C01819=1016.090,-13.127,392.870,165.816,56.691,160.189
C01820=1016.085,-13.376,392.883,165.813,56.699,160.190
C01821=1016.079,-13.625,392.895,165.811,56.706,160.191
C01822=1016.074,-13.876,392.908,165.808,56.714,160.192
C01823=1016.069,-14.125,392.920,165.806,56.722,160.192
C01824=1016.064,-14.374,392.933,165.803,56.729,160.193
C01825=1016.059,-14.625,392.945,165.801,56.737,160.194
C01826=1016.053,-14.874,392.957,165.797,56.744,160.195
C01827=1016.049,-15.123,392.970,165.795,56.752,160.195
C01828=1016.043,-15.373,392.982,165.792,56.760,160.196
C01829=1016.038,-15.623,392.994,165.790,56.767,160.197
C01830=1016.033,-15.873,393.007,165.787,56.775,160.198
C01831=1016.027,-16.122,393.019,165.784,56.782,160.198
C01832=1016.022,-16.372,393.031,165.782,56.790,160.199
C01833=1016.017,-16.621,393.043,165.779,56.797,160.200
C01834=1016.011,-16.871,393.055,165.776,56.805,160.201
C01835=1016.006,-17.121,393.067,165.773,56.813,160.202
C01836=1016.002,-17.371,393.080,165.771,56.821,160.202
C01837=1015.996,-17.621,393.091,165.769,56.828,160.203
C01838=1015.991,-17.870,393.104,165.766,56.836,160.204
C01839=1015.985,-18.120,393.116,165.764,56.844,160.205
C01840=1015.980,-18.369,393.127,165.760,56.852,160.206
C01841=1015.975,-18.619,393.140,165.758,56.859,160.207
C01842=1015.970,-18.869,393.151,165.755,56.867,160.207
C01843=1015.964,-19.118,393.163,165.753,56.875,160.208
C01844=1015.959,-19.368,393.175,165.751,56.882,160.209
C01845=1015.953,-19.618,393.188,165.747,56.890,160.210
C01846=1015.948,-19.868,393.199,165.744,56.897,160.210
C01847=1015.943,-20.117,393.211,165.742,56.905,160.211
C01848=1015.939,-20.367,393.223,165.739,56.913,160.212
C01849=1015.933,-20.616,393.235,165.737,56.920,160.213
C01850=1015.928,-20.867,393.247,165.734,56.928,160.214
C01851=1015.923,-21.116,393.259,165.732,56.936,160.215
C01852=1015.917,-21.392,393.273,165.729,56.944,160.215
C01853=1015.911,-21.670,393.286,165.726,56.952,160.216
C01854=1015.905,-21.946,393.299,165.722,56.961,160.217
C01855=1015.900,-22.223,393.312,165.719,56.969,160.218
C01856=1015.894,-22.472,393.324,165.717,56.977,160.219
C01857=1015.889,-22.722,393.336,165.714,56.984,160.219
C01858=1015.884,-22.972,393.348,165.712,56.992,160.220
C01859=1015.879,-23.222,393.360,165.709,56.999,160.221
C01860=1015.874,-23.471,393.371,165.707,57.007,160.222
C01861=1015.868,-23.721,393.383,165.704,57.014,160.222
C01862=1015.863,-23.970,393.395,165.701,57.022,160.223
C01863=1015.858,-24.220,393.407,165.699,57.029,160.224
C01864=1015.852,-24.470,393.419,165.696,57.037,160.225
C01865=1015.847,-24.719,393.431,165.693,57.044,160.225
C01866=1015.842,-24.969,393.443,165.690,57.052,160.226
C01867=1015.838,-25.219,393.455,165.688,57.060,160.227
C01868=1015.832,-25.468,393.467,165.685,57.067,160.227
C01869=1015.827,-25.718,393.478,165.682,57.074,160.228
C01870=1015.822,-25.968,393.490,165.680,57.082,160.229
C01871=1015.817,-26.217,393.502,165.677,57.089,160.230
C01872=1015.811,-26.468,393.514,165.675,57.097,160.230
C01873=1015.806,-26.717,393.526,165.672,57.104,160.231
C01874=1015.801,-26.967,393.537,165.669,57.111,160.232
C01875=1015.796,-27.216,393.549,165.667,57.119,160.233
C01876=1015.791,-27.466,393.561,165.664,57.126,160.233
C01877=1015.786,-27.715,393.573,165.662,57.134,160.234
C01878=1015.781,-27.965,393.584,165.659,57.141,160.235
C01879=1015.776,-28.215,393.596,165.655,57.149,160.235
C01880=1015.771,-28.465,393.607,165.653,57.156,160.236
C01881=1015.765,-28.714,393.618,165.651,57.164,160.237
C01882=1015.760,-28.963,393.630,165.648,57.172,160.238
C01883=1015.755,-29.213,393.642,165.645,57.179,160.238
C01884=1015.749,-29.464,393.653,165.643,57.187,160.239
C01885=1015.744,-29.714,393.665,165.639,57.195,160.240
C01886=1015.738,-29.963,393.676,165.637,57.202,160.241
C01887=1015.733,-30.213,393.687,165.634,57.209,160.241
C01888=1015.728,-30.463,393.699,165.632,57.217,160.242
C01889=1015.723,-30.712,393.711,165.629,57.225,160.243
C01890=1015.717,-30.961,393.722,165.627,57.232,160.244
C01891=1015.712,-31.211,393.733,165.624,57.239,160.245
C01892=1015.707,-31.461,393.745,165.621,57.248,160.245
C01893=1015.702,-31.711,393.756,165.618,57.255,160.246
C01894=1015.697,-31.961,393.768,165.615,57.262,160.247
C01895=1015.692,-32.210,393.779,165.613,57.270,160.247
C01896=1015.687,-32.460,393.790,165.611,57.278,160.248
C01897=1015.682,-32.710,393.801,165.608,57.285,160.249
C01898=1015.677,-32.959,393.813,165.605,57.292,160.250
C01899=1015.671,-33.209,393.824,165.602,57.299,160.250
C01900=1015.666,-33.459,393.835,165.600,57.307,160.251
C01901=1015.661,-33.709,393.847,165.597,57.315,160.252
C01902=1015.656,-33.958,393.858,165.594,57.322,160.252
C01903=1015.650,-34.208,393.869,165.591,57.330,160.253
C01904=1015.645,-34.458,393.881,165.589,57.337,160.254
C01905=1015.641,-34.707,393.892,165.586,57.345,160.255
C01906=1015.636,-34.957,393.903,165.583,57.352,160.255
C01907=1015.631,-35.206,393.915,165.581,57.359,160.256
C01908=1015.625,-35.456,393.926,165.578,57.366,160.257
C01909=1015.620,-35.706,393.937,165.576,57.374,160.257
C01910=1015.615,-35.955,393.948,165.573,57.381,160.258
C01911=1015.610,-36.205,393.960,165.570,57.389,160.259
C01912=1015.604,-36.455,393.971,165.567,57.396,160.259
C01913=1015.599,-36.705,393.982,165.565,57.403,160.260
C01914=1015.594,-36.954,393.994,165.562,57.410,160.261
C01915=1015.589,-37.204,394.005,165.560,57.418,160.262
C01916=1015.584,-37.445,394.015,165.557,57.425,160.262
C01917=1015.579,-37.685,394.027,165.554,57.432,160.263
C01918=1015.575,-37.925,394.037,165.551,57.439,160.263
C01919=1015.570,-38.166,394.048,165.549,57.447,160.264
C01920=1015.564,-38.406,394.059,165.547,57.453,160.265
C01921=1015.560,-38.647,394.070,165.544,57.460,160.266
C01922=1015.555,-38.887,394.080,165.541,57.467,160.266
C01923=1015.550,-39.128,394.092,165.538,57.474,160.267
C01924=1015.545,-39.378,394.102,165.536,57.482,160.267
C01925=1015.540,-39.627,394.113,165.533,57.489,160.268
C01926=1015.534,-39.877,394.124,165.531,57.497,160.269
C01927=1015.529,-40.127,394.136,165.528,57.504,160.269
C01928=1015.524,-40.376,394.146,165.526,57.512,160.270
C01929=1015.519,-40.626,394.157,165.523,57.519,160.271
C01930=1015.514,-40.875,394.168,165.520,57.526,160.272
C01931=1015.509,-41.126,394.179,165.517,57.535,160.272
C01932=1015.503,-41.375,394.190,165.514,57.542,160.273
C01933=1015.499,-41.624,394.201,165.512,57.549,160.274
C01934=1015.493,-41.874,394.212,165.509,57.556,160.274
C01935=1015.488,-42.124,394.222,165.507,57.564,160.275
C01936=1015.483,-42.374,394.233,165.504,57.571,160.276
C01937=1015.478,-42.624,394.244,165.501,57.579,160.277
C01938=1015.473,-42.873,394.254,165.498,57.586,160.277
C01939=1015.468,-43.123,394.266,165.496,57.593,160.278
C01940=1015.462,-43.373,394.276,165.493,57.601,160.279
C01941=1015.457,-43.623,394.288,165.490,57.608,160.279
C01942=1015.452,-43.872,394.298,165.488,57.615,160.280
C01943=1015.448,-44.122,394.309,165.484,57.623,160.280
C01944=1015.441,-44.416,394.322,165.481,57.632,160.281
C01945=1015.435,-44.711,394.335,165.478,57.640,160.282
C01946=1015.430,-45.005,394.347,165.475,57.649,160.283
C01947=1015.423,-45.299,394.360,165.472,57.657,160.284
C01948=1015.418,-45.549,394.370,165.470,57.665,160.284
C01949=1015.413,-45.798,394.381,165.467,57.672,160.285
C01950=1015.408,-46.048,394.392,165.464,57.679,160.286
C01951=1015.403,-46.298,394.403,165.462,57.687,160.286
C01952=1015.397,-46.548,394.413,165.459,57.694,160.287
C01953=1015.392,-46.797,394.424,165.456,57.701,160.288
C01954=1015.388,-47.047,394.435,165.454,57.708,160.288
C01955=1015.382,-47.297,394.445,165.451,57.715,160.289
C01956=1015.377,-47.546,394.457,165.448,57.722,160.290
C01957=1015.372,-47.796,394.467,165.445,57.729,160.290
C01958=1015.367,-48.046,394.478,165.443,57.737,160.291
C01959=1015.362,-48.295,394.488,165.440,57.744,160.292
C01960=1015.357,-48.545,394.499,165.437,57.751,160.292
C01961=1015.352,-48.795,394.510,165.434,57.758,160.293
C01962=1015.348,-49.045,394.520,165.432,57.766,160.294
C01963=1015.342,-49.294,394.531,165.429,57.773,160.294
C01964=1015.337,-49.544,394.542,165.426,57.780,160.295
C01965=1015.332,-49.793,394.552,165.423,57.787,160.295
C01966=1015.327,-50.044,394.563,165.420,57.794,160.296
C01967=1015.322,-50.293,394.574,165.418,57.802,160.297
C01968=1015.318,-50.543,394.584,165.415,57.809,160.297
C01969=1015.312,-50.792,394.595,165.412,57.816,160.298
C01970=1015.307,-51.043,394.606,165.409,57.823,160.298
C01971=1015.302,-51.292,394.616,165.407,57.830,160.299
C01972=1015.297,-51.542,394.626,165.404,57.838,160.300
C01973=1015.291,-51.792,394.637,165.402,57.845,160.300
C01974=1015.286,-52.041,394.646,165.399,57.853,160.301
C01975=1015.281,-52.291,394.657,165.396,57.860,160.302
C01976=1015.275,-52.541,394.667,165.394,57.868,160.303
C01977=1015.271,-52.791,394.677,165.391,57.875,160.303
C01978=1015.265,-53.041,394.687,165.388,57.882,160.304
C01979=1015.260,-53.290,394.697,165.386,57.889,160.305
C01980=1015.255,-53.566,394.708,165.383,57.898,160.305
C01981=1015.249,-53.842,394.720,165.380,57.906,160.306
C01982=1015.243,-54.118,394.730,165.376,57.914,160.306
C01983=1015.238,-54.394,394.742,165.374,57.922,160.307
C01984=1015.232,-54.644,394.752,165.371,57.929,160.308
C01985=1015.227,-54.894,394.762,165.367,57.936,160.308
C01986=1015.222,-55.144,394.772,165.365,57.944,160.309
C01987=1015.217,-55.394,394.782,165.362,57.951,160.310
C01988=1015.212,-55.643,394.792,165.359,57.958,160.310
C01989=1015.206,-55.894,394.802,165.357,57.966,160.311
C01990=1015.201,-56.143,394.812,165.354,57.973,160.312
C01991=1015.196,-56.393,394.822,165.351,57.980,160.312
C01992=1015.191,-56.642,394.833,165.349,57.987,160.313
C01993=1015.185,-56.892,394.843,165.346,57.995,160.314
C01994=1015.181,-57.141,394.853,165.343,58.002,160.314
C01995=1015.175,-57.391,394.863,165.341,58.009,160.315
C01996=1015.170,-57.641,394.873,165.338,58.016,160.315
C01997=1015.165,-57.891,394.883,165.335,58.023,160.316
C01998=1015.160,-58.140,394.893,165.333,58.031,160.317
C01999=1015.155,-58.391,394.904,165.330,58.038,160.317
C02000=1015.151,-58.640,394.913,165.327,58.045,160.318
C02001=1015.146,-58.890,394.923,165.324,58.052,160.318
C02002=1015.140,-59.140,394.933,165.321,58.059,160.319
C02003=1015.135,-59.389,394.943,165.319,58.067,160.320
C02004=1015.130,-59.639,394.953,165.316,58.074,160.320
C02005=1015.125,-59.889,394.963,165.314,58.081,160.321
C02006=1015.120,-60.139,394.973,165.311,58.088,160.322
C02007=1015.115,-60.388,394.983,165.308,58.096,160.322
C02008=1015.109,-60.638,394.993,165.305,58.103,160.323
C02009=1015.105,-60.888,395.003,165.302,58.110,160.323
C02010=1015.100,-61.137,395.013,165.299,58.117,160.324
C02011=1015.095,-61.388,395.022,165.298,58.123,160.325
C02012=1015.090,-61.637,395.032,165.295,58.130,160.325
C02013=1015.084,-61.887,395.042,165.292,58.138,160.326
C02014=1015.080,-62.137,395.052,165.289,58.145,160.326
C02015=1015.075,-62.386,395.062,165.286,58.152,160.327
C02016=1015.069,-62.636,395.072,165.284,58.159,160.327
C02017=1015.064,-62.886,395.082,165.281,58.166,160.328
C02018=1015.059,-63.136,395.092,165.278,58.173,160.328
C02019=1015.054,-63.385,395.102,165.275,58.180,160.329
C02020=1015.049,-63.635,395.111,165.272,58.187,160.330
C02021=1015.044,-63.885,395.121,165.270,58.194,160.330
C02022=1015.039,-64.135,395.131,165.268,58.201,160.331
C02023=1015.035,-64.384,395.140,165.265,58.208,160.331
C02024=1015.029,-64.634,395.151,165.262,58.215,160.332
C02025=1015.024,-64.884,395.160,165.259,58.222,160.333
C02026=1015.019,-65.133,395.170,165.257,58.229,160.333
C02027=1015.015,-65.384,395.180,165.254,58.236,160.334
C02028=1015.010,-65.633,395.190,165.251,58.243,160.334
C02029=1015.005,-65.883,395.200,165.249,58.249,160.335
C02030=1015.000,-66.133,395.210,165.246,58.256,160.335
C02031=1014.995,-66.382,395.220,165.243,58.263,160.336
C02032=1014.991,-66.632,395.229,165.240,58.270,160.336
C02033=1014.986,-66.882,395.239,165.238,58.278,160.337
C02034=1014.980,-67.132,395.249,165.235,58.285,160.338
C02035=1014.976,-67.381,395.259,165.232,58.291,160.338
C02036=1014.971,-67.631,395.268,165.230,58.298,160.339
C02037=1014.966,-67.882,395.278,165.227,58.305,160.339
C02038=1014.961,-68.131,395.288,165.224,58.312,160.340
C02039=1014.956,-68.380,395.297,165.221,58.319,160.340
C02040=1014.951,-68.630,395.307,165.219,58.325,160.341
C02041=1014.946,-68.880,395.317,165.216,58.332,160.341
C02042=1014.941,-69.130,395.327,165.213,58.339,160.342
C02043=1014.936,-69.379,395.336,165.210,58.345,160.342
C02044=1014.931,-69.656,395.347,165.208,58.353,160.343
C02045=1014.926,-69.934,395.358,165.205,58.360,160.343
C02046=1014.920,-70.210,395.368,165.201,58.368,160.344
C02047=1014.914,-70.488,395.379,165.199,58.376,160.345
C02048=1014.909,-70.738,395.388,165.196,58.382,160.345
C02049=1014.905,-70.987,395.398,165.193,58.389,160.346
C02050=1014.900,-71.237,395.408,165.191,58.396,160.346
C02051=1014.895,-71.487,395.417,165.188,58.402,160.347
C02052=1014.890,-71.737,395.427,165.185,58.409,160.347
C02053=1014.885,-71.987,395.436,165.183,58.416,160.348
C02054=1014.881,-72.236,395.446,165.180,58.422,160.348
C02055=1014.876,-72.486,395.456,165.177,58.430,160.349
C02056=1014.871,-72.736,395.465,165.175,58.435,160.349
C02057=1014.866,-72.986,395.475,165.172,58.443,160.350
C02058=1014.861,-73.235,395.485,165.169,58.450,160.350
C02059=1014.856,-73.485,395.494,165.166,58.456,160.350
C02060=1014.852,-73.735,395.504,165.164,58.463,160.351
C02061=1014.847,-73.985,395.513,165.161,58.469,160.352
C02062=1014.842,-74.234,395.523,165.159,58.476,160.352
C02063=1014.837,-74.483,395.532,165.156,58.482,160.353
C02064=1014.832,-74.734,395.542,165.153,58.489,160.353
C02065=1014.828,-74.984,395.551,165.149,58.496,160.353
C02066=1014.823,-75.234,395.561,165.148,58.502,160.354
C02067=1014.818,-75.484,395.570,165.145,58.509,160.355
C02068=1014.813,-75.733,395.579,165.142,58.517,160.355
C02069=1014.808,-75.983,395.588,165.139,58.523,160.355
C02070=1014.804,-76.233,395.597,165.137,58.530,160.356
C02071=1014.798,-76.482,395.606,165.134,58.537,160.357
C02072=1014.794,-76.732,395.615,165.131,58.543,160.357
///RCONF 1,0,0,0,1,0,0,0,0,0,0,0,0,0,0,0,0,0,0,0,0,0,0,0
C02073=1014.789,-76.982,395.624,165.128,58.550,160.358
C02074=1014.783,-77.232,395.634,165.126,58.557,160.358
C02075=1014.778,-77.482,395.643,165.123,58.563,160.359
C02076=1014.774,-77.732,395.652,165.120,58.570,160.359
C02077=1014.769,-77.981,395.662,165.117,58.577,160.359
C02078=1014.764,-78.231,395.670,165.115,58.583,160.360
C02079=1014.759,-78.481,395.680,165.113,58.591,160.361
C02080=1014.754,-78.730,395.689,165.109,58.597,160.361
C02081=1014.749,-78.980,395.698,165.107,58.604,160.362
C02082=1014.745,-79.230,395.707,165.104,58.610,160.362
C02083=1014.740,-79.480,395.716,165.101,58.617,160.363
C02084=1014.735,-79.729,395.725,165.098,58.624,160.363
C02085=1014.730,-79.979,395.734,165.096,58.630,160.364
C02086=1014.725,-80.229,395.743,165.093,58.637,160.364
C02087=1014.721,-80.479,395.752,165.090,58.644,160.364
C02088=1014.716,-80.729,395.761,165.089,58.650,160.365
C02089=1014.710,-80.979,395.769,165.085,58.657,160.365
C02090=1014.706,-81.229,395.778,165.082,58.664,160.366
C02091=1014.700,-81.478,395.788,165.080,58.671,160.367
C02092=1014.696,-81.728,395.797,165.076,58.677,160.367
C02093=1014.691,-81.977,395.805,165.075,58.684,160.368
C02094=1014.685,-82.227,395.814,165.072,58.691,160.368
C02095=1014.681,-82.477,395.823,165.068,58.698,160.368
C02096=1014.675,-82.727,395.831,165.066,58.705,160.369
C02097=1014.671,-82.977,395.840,165.063,58.711,160.369
C02098=1014.666,-83.227,395.849,165.061,58.718,160.370
C02099=1014.661,-83.477,395.858,165.058,58.725,160.371
C02100=1014.656,-83.726,395.866,165.056,58.731,160.371
C02101=1014.651,-83.976,395.875,165.053,58.738,160.372
C02102=1014.646,-84.226,395.884,165.050,58.745,160.372
C02103=1014.641,-84.476,395.892,165.047,58.752,160.372
C02104=1014.636,-84.726,395.902,165.045,58.758,160.373
C02105=1014.632,-84.975,395.910,165.042,58.765,160.373
C02106=1014.626,-85.225,395.918,165.038,58.771,160.374
C02107=1014.622,-85.475,395.927,165.037,58.778,160.374
C02108=1014.616,-85.754,395.937,165.033,58.786,160.375
C02109=1014.611,-86.033,395.947,165.030,58.793,160.375
C02110=1014.605,-86.312,395.956,165.028,58.800,160.376
C02111=1014.600,-86.591,395.966,165.024,58.807,160.376
C02112=1014.595,-86.841,395.975,165.022,58.814,160.377
C02113=1014.590,-87.091,395.983,165.019,58.821,160.377
C02114=1014.585,-87.341,395.991,165.015,58.827,160.377
C02115=1014.581,-87.590,396.000,165.014,58.834,160.378
C02116=1014.576,-87.840,396.008,165.010,58.840,160.378
C02117=1014.571,-88.090,396.017,165.009,58.847,160.379
C02118=1014.566,-88.340,396.026,165.005,58.853,160.379
C02119=1014.561,-88.590,396.034,165.002,58.860,160.380
C02120=1014.556,-88.840,396.044,165.000,58.866,160.380
C02121=1014.551,-89.089,396.052,164.997,58.873,160.381
C02122=1014.547,-89.339,396.061,164.995,58.879,160.381
C02123=1014.542,-89.589,396.068,164.992,58.886,160.382
C02124=1014.537,-89.839,396.077,164.990,58.892,160.382
C02125=1014.532,-90.089,396.086,164.986,58.898,160.382
C02126=1014.527,-90.338,396.094,164.983,58.905,160.383
C02127=1014.523,-90.588,396.103,164.981,58.911,160.383
C02128=1014.518,-90.837,396.112,164.978,58.918,160.384
C02129=1014.513,-91.088,396.119,164.976,58.924,160.384
C02130=1014.508,-91.338,396.129,164.973,58.930,160.384
C02131=1014.504,-91.587,396.137,164.971,58.937,160.385
C02132=1014.499,-91.837,396.146,164.968,58.943,160.385
C02133=1014.494,-92.087,396.154,164.965,58.949,160.386
C02134=1014.489,-92.337,396.162,164.962,58.956,160.386
C02135=1014.485,-92.586,396.171,164.960,58.962,160.387
C02136=1014.480,-92.836,396.179,164.957,58.969,160.387
C02137=1014.475,-93.086,396.188,164.955,58.975,160.388
C02138=1014.470,-93.336,396.196,164.951,58.981,160.388
C02139=1014.465,-93.585,396.204,164.949,58.987,160.388
C02140=1014.461,-93.835,396.213,164.947,58.993,160.389
C02141=1014.456,-94.086,396.221,164.944,59.000,160.389
C02142=1014.452,-94.335,396.230,164.941,59.006,160.389
C02143=1014.447,-94.585,396.238,164.938,59.012,160.390
C02144=1014.442,-94.834,396.247,164.936,59.018,160.390
C02145=1014.438,-95.084,396.255,164.933,59.025,160.391
C02146=1014.433,-95.334,396.263,164.931,59.031,160.391
C02147=1014.427,-95.584,396.272,164.928,59.037,160.392
C02148=1014.423,-95.834,396.280,164.925,59.044,160.392
C02149=1014.418,-96.083,396.288,164.923,59.050,160.392
C02150=1014.414,-96.334,396.297,164.920,59.056,160.393
C02151=1014.410,-96.583,396.305,164.917,59.062,160.393
C02152=1014.404,-96.833,396.313,164.915,59.068,160.393
C02153=1014.400,-97.083,396.322,164.912,59.074,160.394
C02154=1014.395,-97.333,396.330,164.909,59.080,160.394
C02155=1014.391,-97.583,396.339,164.907,59.086,160.395
C02156=1014.386,-97.833,396.346,164.903,59.092,160.394
C02157=1014.381,-98.082,396.355,164.901,59.098,160.395
C02158=1014.376,-98.332,396.362,164.898,59.105,160.396
C02159=1014.372,-98.582,396.371,164.896,59.111,160.396
C02160=1014.367,-98.832,396.379,164.893,59.118,160.396
C02161=1014.362,-99.082,396.387,164.890,59.124,160.397
C02162=1014.357,-99.332,396.395,164.888,59.130,160.397
C02163=1014.353,-99.581,396.403,164.885,59.136,160.397
C02164=1014.348,-99.831,396.411,164.883,59.142,160.398
C02165=1014.343,-100.081,396.418,164.879,59.149,160.398
C02166=1014.338,-100.331,396.427,164.877,59.155,160.399
C02167=1014.334,-100.580,396.434,164.874,59.161,160.399
C02168=1014.328,-100.830,396.443,164.872,59.167,160.399
C02169=1014.324,-101.081,396.451,164.869,59.173,160.400
C02170=1014.320,-101.330,396.459,164.866,59.179,160.400
C02171=1014.315,-101.580,396.467,164.864,59.185,160.400
C02172=1014.310,-101.861,396.475,164.861,59.193,160.401
C02173=1014.304,-102.142,396.484,164.858,59.199,160.401
C02174=1014.299,-102.423,396.493,164.855,59.206,160.402
C02175=1014.293,-102.704,396.502,164.852,59.213,160.402
C02176=1014.288,-102.953,396.510,164.850,59.219,160.402
C02177=1014.284,-103.204,396.518,164.846,59.225,160.403
C02178=1014.279,-103.453,396.525,164.844,59.231,160.403
C02179=1014.275,-103.703,396.534,164.842,59.237,160.404
C02180=1014.270,-103.953,396.542,164.838,59.244,160.404
C02181=1014.265,-104.203,396.550,164.836,59.250,160.404
C02182=1014.261,-104.453,396.557,164.834,59.256,160.405
C02183=1014.256,-104.703,396.565,164.831,59.262,160.405
C02184=1014.251,-104.952,396.573,164.828,59.267,160.405
C02185=1014.246,-105.203,396.581,164.826,59.273,160.405
C02186=1014.242,-105.452,396.588,164.822,59.280,160.406
C02187=1014.237,-105.702,396.596,164.820,59.286,160.406
C02188=1014.232,-105.952,396.604,164.818,59.292,160.407
C02189=1014.228,-106.201,396.611,164.816,59.298,160.407
C02190=1014.223,-106.452,396.619,164.812,59.304,160.407
C02191=1014.218,-106.701,396.627,164.809,59.310,160.407
C02192=1014.213,-106.951,396.635,164.807,59.316,160.408
C02193=1014.209,-107.201,396.642,164.805,59.322,160.408
C02194=1014.204,-107.451,396.650,164.801,59.327,160.408
C02195=1014.200,-107.701,396.657,164.799,59.333,160.409
C02196=1014.195,-107.950,396.665,164.797,59.339,160.409
C02197=1014.190,-108.201,396.673,164.794,59.345,160.410
C02198=1014.186,-108.450,396.681,164.792,59.351,160.410
C02199=1014.181,-108.700,396.689,164.788,59.357,160.410
C02200=1014.176,-108.950,396.696,164.786,59.363,160.410
C02201=1014.172,-109.199,396.703,164.784,59.369,160.411
C02202=1014.167,-109.450,396.711,164.781,59.375,160.411
C02203=1014.163,-109.699,396.719,164.778,59.381,160.411
C02204=1014.158,-109.950,396.726,164.775,59.387,160.412
C02205=1014.153,-110.199,396.733,164.773,59.393,160.412
C02206=1014.148,-110.448,396.741,164.771,59.399,160.413
C02207=1014.143,-110.699,396.748,164.767,59.405,160.413
C02208=1014.139,-110.948,396.756,164.765,59.411,160.413
C02209=1014.135,-111.198,396.763,164.763,59.417,160.413
C02210=1014.130,-111.448,396.771,164.760,59.422,160.414
C02211=1014.125,-111.698,396.778,164.757,59.428,160.414
C02212=1014.121,-111.948,396.786,164.755,59.434,160.415
C02213=1014.115,-112.198,396.793,164.751,59.440,160.414
C02214=1014.111,-112.447,396.800,164.749,59.446,160.415
C02215=1014.107,-112.697,396.808,164.747,59.452,160.415
C02216=1014.102,-112.947,396.815,164.744,59.457,160.415
C02217=1014.097,-113.197,396.823,164.742,59.463,160.416
C02218=1014.093,-113.447,396.830,164.739,59.468,160.416
C02219=1014.089,-113.697,396.837,164.737,59.474,160.416
C02220=1014.084,-113.947,396.845,164.734,59.480,160.417
C02221=1014.080,-114.197,396.852,164.732,59.486,160.417
C02222=1014.075,-114.446,396.859,164.728,59.492,160.417
C02223=1014.070,-114.696,396.867,164.726,59.497,160.417
C02224=1014.065,-114.946,396.874,164.723,59.503,160.418
C02225=1014.061,-115.196,396.881,164.720,59.509,160.418
C02226=1014.056,-115.445,396.889,164.718,59.515,160.418
C02227=1014.051,-115.696,396.895,164.715,59.520,160.419
C02228=1014.047,-115.946,396.903,164.713,59.526,160.419
C02229=1014.042,-116.195,396.910,164.710,59.531,160.419
C02230=1014.038,-116.445,396.918,164.708,59.537,160.420
C02231=1014.032,-116.695,396.925,164.705,59.543,160.420
C02232=1014.028,-116.945,396.931,164.703,59.549,160.420
C02233=1014.024,-117.195,396.939,164.700,59.554,160.420
C02234=1014.020,-117.444,396.946,164.698,59.560,160.421
C02235=1014.014,-117.694,396.953,164.695,59.565,160.421
C02236=1014.009,-117.976,396.961,164.692,59.572,160.421
C02237=1014.004,-118.257,396.969,164.689,59.578,160.421
C02238=1013.999,-118.538,396.977,164.686,59.584,160.422
C02239=1013.994,-118.819,396.985,164.683,59.591,160.422
C02240=1013.989,-119.069,396.992,164.681,59.597,160.422
C02241=1013.985,-119.320,396.999,164.678,59.602,160.423
C02242=1013.980,-119.569,397.006,164.676,59.608,160.423
C02243=1013.975,-119.819,397.014,164.673,59.613,160.423
C02244=1013.971,-120.069,397.020,164.670,59.619,160.423
C02245=1013.966,-120.318,397.027,164.668,59.625,160.424
C02246=1013.962,-120.568,397.034,164.665,59.630,160.424
C02247=1013.957,-120.819,397.041,164.663,59.636,160.424
C02248=1013.953,-121.068,397.049,164.660,59.641,160.424
C02249=1013.948,-121.318,397.055,164.657,59.647,160.425
C02250=1013.944,-121.568,397.062,164.655,59.653,160.425
C02251=1013.939,-121.818,397.070,164.652,59.658,160.425
C02252=1013.935,-122.068,397.076,164.649,59.663,160.425
C02253=1013.930,-122.317,397.083,164.648,59.669,160.426
C02254=1013.926,-122.567,397.090,164.645,59.674,160.426
C02255=1013.921,-122.817,397.097,164.643,59.679,160.426
C02256=1013.916,-123.067,397.105,164.640,59.685,160.426
C02257=1013.912,-123.317,397.111,164.638,59.691,160.427
C02258=1013.907,-123.567,397.118,164.635,59.696,160.427
C02259=1013.903,-123.817,397.125,164.632,59.701,160.427
C02260=1013.898,-124.066,397.132,164.629,59.707,160.427
C02261=1013.894,-124.317,397.138,164.627,59.711,160.428
C02262=1013.889,-124.566,397.146,164.625,59.717,160.428
C02263=1013.885,-124.816,397.152,164.622,59.723,160.428
C02264=1013.880,-125.066,397.159,164.619,59.728,160.428
C02265=1013.876,-125.316,397.166,164.617,59.733,160.428
C02266=1013.871,-125.565,397.173,164.614,59.739,160.429
C02267=1013.867,-125.816,397.179,164.612,59.745,160.429
C02268=1013.862,-126.066,397.185,164.609,59.750,160.429
C02269=1013.858,-126.315,397.193,164.607,59.755,160.429
C02270=1013.853,-126.565,397.199,164.604,59.760,160.430
C02271=1013.849,-126.815,397.206,164.602,59.766,160.430
C02272=1013.844,-127.065,397.212,164.599,59.771,160.430
C02273=1013.840,-127.315,397.219,164.596,59.777,160.430
C02274=1013.835,-127.564,397.226,164.595,59.782,160.431
C02275=1013.831,-127.814,397.233,164.592,59.787,160.431
C02276=1013.826,-128.064,397.239,164.589,59.792,160.431
C02277=1013.822,-128.314,397.246,164.586,59.797,160.431
C02278=1013.818,-128.563,397.253,164.584,59.802,160.431
C02279=1013.813,-128.813,397.261,164.582,59.806,160.431
C02280=1013.810,-129.062,397.270,164.580,59.810,160.431
C02281=1013.807,-129.312,397.279,164.578,59.813,160.431
C02282=1013.804,-129.562,397.288,164.575,59.817,160.431
C02283=1013.802,-129.812,397.299,164.572,59.819,160.431
C02284=1013.799,-130.061,397.310,164.570,59.821,160.430
C02285=1013.798,-130.311,397.321,164.568,59.821,160.430
C02286=1013.797,-130.560,397.334,164.566,59.822,160.429
C02287=1013.796,-130.810,397.347,164.563,59.822,160.429
C02288=1013.795,-131.060,397.360,164.561,59.822,160.428
C02289=1013.795,-131.310,397.374,164.560,59.822,160.427
C02290=1013.794,-131.559,397.388,164.557,59.821,160.426
C02291=1013.795,-131.809,397.403,164.555,59.819,160.425
C02292=1013.796,-132.059,397.419,164.552,59.817,160.424
C02293=1013.797,-132.308,397.435,164.551,59.814,160.423
C02294=1013.798,-132.558,397.452,164.549,59.811,160.422
C02295=1013.800,-132.807,397.470,164.547,59.808,160.421
C02296=1013.802,-133.057,397.488,164.545,59.803,160.419
C02297=1013.804,-133.307,397.507,164.543,59.799,160.418
C02298=1013.807,-133.556,397.527,164.541,59.794,160.416
C02299=1013.810,-133.806,397.547,164.539,59.788,160.415
C02300=1013.579,-133.832,397.130,164.519,60.110,160.468
C02301=1013.576,-133.583,397.110,164.521,60.115,160.470
C02302=1013.574,-133.333,397.091,164.523,60.119,160.471
C02303=1013.571,-133.083,397.072,164.526,60.124,160.473
C02304=1013.570,-132.833,397.053,164.527,60.128,160.474
C02305=1013.568,-132.584,397.035,164.530,60.131,160.475
C02306=1013.566,-132.334,397.018,164.530,60.134,160.476
C02307=1013.565,-132.084,397.003,164.533,60.137,160.478
C02308=1013.564,-131.835,396.986,164.535,60.139,160.478
C02309=1013.564,-131.585,396.971,164.538,60.140,160.480
C02310=1013.564,-131.336,396.957,164.539,60.142,160.480
C02311=1013.565,-131.086,396.943,164.541,60.142,160.481
C02312=1013.565,-130.836,396.929,164.544,60.142,160.482
C02313=1013.566,-130.587,396.917,164.545,60.142,160.482
C02314=1013.568,-130.338,396.904,164.548,60.141,160.483
C02315=1013.569,-130.088,396.893,164.550,60.140,160.483
C02316=1013.571,-129.838,396.881,164.552,60.138,160.484
C02317=1013.574,-129.588,396.871,164.554,60.137,160.484
C02318=1013.576,-129.338,396.862,164.558,60.134,160.485
C02319=1013.579,-129.088,396.852,164.560,60.131,160.485
C02320=1013.583,-128.839,396.844,164.562,60.127,160.485
C02321=1013.586,-128.590,396.836,164.563,60.123,160.484
C02322=1013.590,-128.340,396.829,164.567,60.119,160.485
C02323=1013.595,-128.090,396.822,164.568,60.114,160.484
C02324=1013.600,-127.841,396.815,164.571,60.109,160.484
C02325=1013.604,-127.591,396.809,164.574,60.104,160.484
C02326=1013.608,-127.342,396.802,164.576,60.099,160.484
C02327=1013.613,-127.092,396.796,164.579,60.094,160.484
C02328=1013.617,-126.842,396.789,164.581,60.089,160.484
C02329=1013.622,-126.592,396.782,164.584,60.084,160.483
C02330=1013.626,-126.342,396.776,164.587,60.078,160.483
C02331=1013.631,-126.092,396.770,164.588,60.073,160.483
C02332=1013.635,-125.842,396.762,164.591,60.068,160.483
C02333=1013.640,-125.593,396.756,164.594,60.063,160.483
C02334=1013.644,-125.342,396.749,164.597,60.058,160.483
C02335=1013.648,-125.093,396.742,164.598,60.053,160.482
C02336=1013.653,-124.843,396.736,164.601,60.047,160.482
C02337=1013.658,-124.593,396.728,164.604,60.042,160.482
C02338=1013.662,-124.343,396.722,164.606,60.037,160.482
C02339=1013.667,-124.093,396.715,164.608,60.032,160.481
C02340=1013.671,-123.843,396.708,164.611,60.027,160.481
C02341=1013.677,-123.593,396.701,164.613,60.022,160.481
C02342=1013.681,-123.343,396.694,164.616,60.016,160.481
C02343=1013.685,-123.093,396.687,164.619,60.011,160.481
C02344=1013.690,-122.843,396.681,164.621,60.006,160.481
C02345=1013.694,-122.594,396.673,164.623,60.001,160.480
C02346=1013.698,-122.343,396.667,164.626,59.996,160.480
C02347=1013.703,-122.094,396.660,164.629,59.990,160.480
C02348=1013.707,-121.844,396.653,164.632,59.985,160.480
C02349=1013.712,-121.594,396.646,164.633,59.980,160.479
C02350=1013.716,-121.344,396.640,164.636,59.975,160.479
C02351=1013.721,-121.095,396.632,164.638,59.969,160.479
C02352=1013.725,-120.845,396.625,164.641,59.963,160.479
C02353=1013.731,-120.594,396.619,164.644,59.958,160.479
C02354=1013.735,-120.345,396.611,164.646,59.953,160.478
C02355=1013.739,-120.095,396.604,164.648,59.948,160.478
C02356=1013.744,-119.845,396.598,164.651,59.943,160.478
C02357=1013.748,-119.596,396.590,164.654,59.937,160.478
C02358=1013.752,-119.345,396.584,164.656,59.931,160.477
C02359=1013.757,-119.096,396.576,164.659,59.926,160.477
C02360=1013.762,-118.846,396.569,164.662,59.921,160.477
C02361=1013.766,-118.565,396.562,164.664,59.915,160.477
C02362=1013.772,-118.283,396.553,164.667,59.908,160.476
C02363=1013.778,-118.002,396.546,164.670,59.903,160.476
C02364=1013.783,-117.721,396.537,164.673,59.896,160.476
C02365=1013.787,-117.471,396.530,164.675,59.891,160.476
C02366=1013.792,-117.222,396.523,164.677,59.885,160.475
C02367=1013.796,-116.972,396.517,164.680,59.880,160.475
C02368=1013.800,-116.722,396.509,164.683,59.875,160.475
C02369=1013.805,-116.472,396.501,164.685,59.869,160.475
C02370=1013.810,-116.222,396.494,164.688,59.863,160.474
C02371=1013.815,-115.972,396.488,164.690,59.858,160.474
C02372=1013.819,-115.723,396.481,164.693,59.853,160.474
C02373=1013.823,-115.473,396.473,164.695,59.847,160.474
C02374=1013.828,-115.223,396.465,164.698,59.841,160.473
C02375=1013.833,-114.973,396.459,164.700,59.835,160.473
C02376=1013.837,-114.723,396.452,164.703,59.830,160.473
C02377=1013.842,-114.474,396.444,164.706,59.825,160.473
C02378=1013.847,-114.223,396.437,164.708,59.819,160.472
C02379=1013.851,-113.974,396.429,164.711,59.813,160.472
C02380=1013.855,-113.724,396.422,164.714,59.808,160.472
C02381=1013.860,-113.475,396.415,164.716,59.802,160.471
C02382=1013.865,-113.224,396.408,164.719,59.797,160.471
C02383=1013.869,-112.974,396.401,164.722,59.791,160.471
C02384=1013.874,-112.724,396.393,164.724,59.785,160.471
C02385=1013.878,-112.475,396.386,164.727,59.780,160.471
C02386=1013.883,-112.224,396.378,164.729,59.774,160.470
C02387=1013.887,-111.975,396.371,164.732,59.769,160.470
C02388=1013.892,-111.725,396.363,164.734,59.763,160.469
C02389=1013.896,-111.475,396.356,164.737,59.757,160.469
C02390=1013.902,-111.225,396.349,164.739,59.751,160.469
C02391=1013.906,-110.976,396.341,164.742,59.746,160.469
C02392=1013.911,-110.726,396.334,164.744,59.740,160.468
C02393=1013.916,-110.476,396.326,164.747,59.735,160.468
C02394=1013.920,-110.226,396.319,164.749,59.729,160.468
C02395=1013.924,-109.977,396.311,164.751,59.723,160.468
C02396=1013.929,-109.726,396.304,164.754,59.717,160.467
C02397=1013.934,-109.477,396.296,164.756,59.712,160.467
C02398=1013.939,-109.227,396.289,164.760,59.705,160.467
C02399=1013.944,-108.977,396.282,164.763,59.700,160.467
C02400=1013.948,-108.727,396.274,164.765,59.694,160.466
C02401=1013.952,-108.478,396.267,164.767,59.688,160.466
C02402=1013.957,-108.227,396.259,164.770,59.683,160.465
C02403=1013.962,-107.978,396.252,164.772,59.677,160.465
C02404=1013.967,-107.727,396.244,164.775,59.671,160.465
C02405=1013.971,-107.478,396.236,164.777,59.665,160.464
C02406=1013.975,-107.228,396.229,164.780,59.659,160.464
C02407=1013.980,-106.978,396.221,164.783,59.654,160.464
C02408=1013.985,-106.728,396.214,164.785,59.648,160.464
C02409=1013.990,-106.478,396.205,164.788,59.642,160.463
C02410=1013.994,-106.229,396.198,164.790,59.636,160.463
C02411=1013.999,-105.979,396.191,164.792,59.630,160.462
C02412=1014.004,-105.729,396.183,164.795,59.625,160.462
C02413=1014.008,-105.479,396.175,164.798,59.619,160.462
C02414=1014.013,-105.229,396.168,164.801,59.612,160.462
C02415=1014.018,-104.980,396.159,164.803,59.607,160.461
C02416=1014.022,-104.729,396.151,164.806,59.601,160.461
C02417=1014.026,-104.480,396.144,164.808,59.595,160.461
C02418=1014.031,-104.230,396.136,164.812,59.589,160.461
C02419=1014.036,-103.980,396.128,164.814,59.583,160.460
C02420=1014.040,-103.731,396.120,164.816,59.577,160.460
C02421=1014.045,-103.480,396.113,164.818,59.571,160.459
C02422=1014.049,-103.231,396.105,164.821,59.566,160.459
C02423=1014.055,-102.981,396.097,164.824,59.560,160.459
C02424=1014.059,-102.731,396.089,164.827,59.554,160.458
C02425=1014.065,-102.450,396.080,164.830,59.547,160.458
C02426=1014.070,-102.169,396.072,164.832,59.540,160.458
C02427=1014.075,-101.889,396.063,164.836,59.533,160.457
C02428=1014.081,-101.607,396.054,164.839,59.527,160.457
C02429=1014.084,-101.357,396.046,164.841,59.521,160.457
C02430=1014.089,-101.107,396.038,164.843,59.515,160.456
C02431=1014.094,-100.858,396.030,164.846,59.509,160.456
C02432=1014.099,-100.608,396.022,164.849,59.502,160.455
C02433=1014.103,-100.358,396.015,164.851,59.496,160.455
C02434=1014.109,-100.108,396.006,164.854,59.491,160.455
C02435=1014.113,-99.859,395.999,164.857,59.485,160.455
C02436=1014.118,-99.609,395.990,164.859,59.478,160.454
C02437=1014.123,-99.359,395.983,164.861,59.472,160.454
C02438=1014.128,-99.109,395.975,164.865,59.466,160.453
C02439=1014.132,-98.859,395.966,164.867,59.460,160.453
C02440=1014.136,-98.609,395.959,164.869,59.454,160.452
C02441=1014.141,-98.359,395.951,164.872,59.447,160.452
C02442=1014.146,-98.110,395.943,164.875,59.441,160.452
C02443=1014.151,-97.860,395.935,164.878,59.435,160.451
C02444=1014.156,-97.610,395.926,164.880,59.429,160.451
C02445=1014.160,-97.360,395.918,164.883,59.424,160.451
C02446=1014.165,-97.110,395.910,164.885,59.418,160.450
C02447=1014.169,-96.861,395.901,164.888,59.411,160.450
C02448=1014.174,-96.611,395.893,164.891,59.405,160.450
C02449=1014.179,-96.361,395.884,164.893,59.399,160.449
C02450=1014.183,-96.111,395.877,164.896,59.393,160.449
C02451=1014.188,-95.861,395.868,164.898,59.387,160.448
C02452=1014.193,-95.611,395.859,164.901,59.381,160.448
C02453=1014.197,-95.362,395.852,164.903,59.375,160.448
C02454=1014.202,-95.112,395.844,164.907,59.369,160.448
C02455=1014.207,-94.862,395.834,164.909,59.363,160.447
C02456=1014.211,-94.612,395.827,164.911,59.357,160.447
C02457=1014.216,-94.362,395.818,164.914,59.350,160.446
C02458=1014.221,-94.113,395.809,164.917,59.344,160.446
C02459=1014.225,-93.863,395.802,164.920,59.338,160.446
C02460=1014.230,-93.613,395.793,164.922,59.332,160.445
C02461=1014.235,-93.363,395.785,164.924,59.326,160.445
C02462=1014.239,-93.113,395.777,164.928,59.320,160.445
C02463=1014.244,-92.864,395.768,164.930,59.314,160.444
C02464=1014.249,-92.614,395.760,164.933,59.307,160.444
C02465=1014.253,-92.365,395.751,164.935,59.301,160.443
C02466=1014.258,-92.114,395.743,164.937,59.295,160.443
C02467=1014.263,-91.864,395.734,164.941,59.289,160.443
C02468=1014.268,-91.614,395.725,164.943,59.283,160.442
C02469=1014.273,-91.365,395.717,164.946,59.276,160.442
C02470=1014.277,-91.115,395.709,164.948,59.269,160.441
C02471=1014.282,-90.865,395.701,164.951,59.263,160.441
C02472=1014.286,-90.616,395.692,164.953,59.257,160.440
C02473=1014.291,-90.366,395.683,164.957,59.251,160.440
C02474=1014.296,-90.116,395.676,164.959,59.245,160.440
C02475=1014.301,-89.866,395.666,164.962,59.238,160.439
C02476=1014.306,-89.617,395.658,164.964,59.232,160.439
C02477=1014.310,-89.367,395.649,164.967,59.225,160.438
C02478=1014.315,-89.117,395.641,164.969,59.219,160.438
C02479=1014.320,-88.867,395.633,164.973,59.212,160.438
C02480=1014.325,-88.617,395.624,164.975,59.206,160.437
C02481=1014.329,-88.368,395.616,164.977,59.199,160.437
C02482=1014.334,-88.118,395.607,164.980,59.193,160.436
C02483=1014.339,-87.868,395.598,164.983,59.187,160.436
C02484=1014.344,-87.618,395.590,164.985,59.181,160.435
C02485=1014.349,-87.367,395.581,164.988,59.174,160.435
C02486=1014.353,-87.118,395.573,164.990,59.168,160.434
C02487=1014.358,-86.868,395.564,164.993,59.161,160.434
C02488=1014.363,-86.619,395.556,164.996,59.154,160.434
C02489=1014.368,-86.340,395.546,164.999,59.148,160.433
C02490=1014.374,-86.060,395.536,165.002,59.140,160.433
C02491=1014.380,-85.782,395.527,165.005,59.133,160.432
C02492=1014.385,-85.503,395.517,165.008,59.126,160.432
C02493=1014.390,-85.253,395.509,165.010,59.119,160.431
C02494=1014.395,-85.003,395.500,165.013,59.112,160.431
C02495=1014.400,-84.754,395.491,165.016,59.105,160.430
C02496=1014.404,-84.504,395.482,165.018,59.099,160.430
C02497=1014.409,-84.255,395.474,165.022,59.093,160.429
C02498=1014.414,-84.005,395.465,165.023,59.086,160.429
C02499=1014.419,-83.755,395.457,165.026,59.080,160.428
C02500=1014.424,-83.505,395.448,165.029,59.072,160.428
C02501=1014.429,-83.255,395.439,165.031,59.066,160.427
C02502=1014.434,-83.005,395.431,165.034,59.059,160.427
C02503=1014.438,-82.755,395.422,165.037,59.053,160.427
C02504=1014.444,-82.506,395.413,165.040,59.046,160.426
C02505=1014.449,-82.256,395.405,165.042,59.040,160.425
C02506=1014.453,-82.006,395.395,165.045,59.033,160.425
C02507=1014.459,-81.756,395.387,165.048,59.026,160.425
C02508=1014.463,-81.507,395.378,165.050,59.019,160.424
C02509=1014.468,-81.257,395.370,165.053,59.012,160.423
C02510=1014.472,-81.007,395.361,165.056,59.006,160.423
C02511=1014.478,-80.757,395.352,165.059,58.999,160.422
C02512=1014.483,-80.508,395.344,165.061,58.993,160.422
C02513=1014.488,-80.258,395.335,165.063,58.985,160.421
C02514=1014.492,-80.008,395.326,165.067,58.979,160.421
C02515=1014.497,-79.758,395.317,165.068,58.972,160.420
C02516=1014.502,-79.508,395.308,165.072,58.966,160.420
C02517=1014.507,-79.259,395.298,165.074,58.959,160.420
C02518=1014.511,-79.008,395.289,165.077,58.953,160.419
C02519=1014.516,-78.759,395.281,165.080,58.946,160.419
C02520=1014.521,-78.509,395.272,165.083,58.939,160.418
C02521=1014.526,-78.259,395.262,165.085,58.933,160.418
C02522=1014.531,-78.010,395.253,165.088,58.926,160.417
C02523=1014.536,-77.760,395.244,165.091,58.920,160.417
C02524=1014.540,-77.510,395.235,165.093,58.913,160.416
C02525=1014.546,-77.260,395.226,165.095,58.906,160.416
C02526=1014.551,-77.010,395.217,165.099,58.899,160.415
C02527=1014.555,-76.760,395.207,165.100,58.893,160.415
C02528=1014.560,-76.510,395.198,165.104,58.886,160.414
C02529=1014.565,-76.261,395.189,165.106,58.879,160.414
C02530=1014.570,-76.011,395.180,165.110,58.873,160.413
C02531=1014.575,-75.761,395.170,165.111,58.866,160.413
C02532=1014.580,-75.511,395.162,165.114,58.859,160.412
///RCONF 1,0,0,0,0,0,0,0,0,0,0,0,0,0,0,0,0,0,0,0,0,0,0,0
C02533=1014.585,-75.261,395.153,165.117,58.852,160.412
C02534=1014.589,-75.012,395.143,165.120,58.845,160.411
C02535=1014.595,-74.762,395.134,165.122,58.838,160.410
C02536=1014.599,-74.512,395.125,165.125,58.832,160.410
C02537=1014.604,-74.263,395.116,165.128,58.825,160.410
C02538=1014.609,-74.013,395.106,165.130,58.819,160.409
C02539=1014.614,-73.763,395.096,165.133,58.812,160.409
C02540=1014.619,-73.513,395.087,165.136,58.805,160.408
C02541=1014.623,-73.263,395.077,165.138,58.799,160.408
C02542=1014.628,-73.014,395.068,165.141,58.792,160.407
C02543=1014.633,-72.764,395.059,165.143,58.786,160.407
C02544=1014.638,-72.514,395.049,165.146,58.779,160.406
C02545=1014.642,-72.264,395.040,165.149,58.772,160.406
C02546=1014.647,-72.015,395.030,165.152,58.766,160.405
C02547=1014.652,-71.764,395.020,165.154,58.759,160.405
C02548=1014.657,-71.515,395.011,165.157,58.753,160.404
C02549=1014.662,-71.265,395.001,165.160,58.745,160.404
C02550=1014.666,-71.015,394.992,165.162,58.739,160.403
C02551=1014.671,-70.766,394.982,165.165,58.732,160.403
C02552=1014.676,-70.517,394.972,165.167,58.725,160.402
C02553=1014.681,-70.239,394.961,165.170,58.718,160.402
C02554=1014.687,-69.962,394.950,165.173,58.711,160.401
C02555=1014.692,-69.685,394.940,165.177,58.703,160.401
C02556=1014.697,-69.409,394.929,165.179,58.695,160.400
C02557=1014.701,-69.159,394.920,165.182,58.689,160.399
C02558=1014.707,-68.908,394.910,165.185,58.682,160.399
C02559=1014.712,-68.659,394.900,165.186,58.675,160.398
C02560=1014.716,-68.409,394.891,165.190,58.669,160.398
C02561=1014.721,-68.160,394.881,165.193,58.662,160.397
C02562=1014.726,-67.909,394.871,165.195,58.655,160.397
C02563=1014.731,-67.659,394.862,165.198,58.649,160.396
C02564=1014.736,-67.410,394.852,165.200,58.642,160.396
C02565=1014.741,-67.161,394.842,165.203,58.634,160.395
C02566=1014.745,-66.911,394.833,165.206,58.627,160.395
C02567=1014.751,-66.661,394.823,165.209,58.620,160.394
C02568=1014.755,-66.411,394.813,165.211,58.614,160.393
C02569=1014.760,-66.162,394.804,165.214,58.607,160.393
C02570=1014.766,-65.912,394.793,165.216,58.600,160.392
C02571=1014.770,-65.662,394.784,165.219,58.593,160.392
C02572=1014.775,-65.412,394.774,165.222,58.586,160.391
C02573=1014.780,-65.163,394.765,165.225,58.579,160.391
C02574=1014.785,-64.913,394.755,165.227,58.573,160.390
C02575=1014.790,-64.663,394.745,165.230,58.566,160.390
C02576=1014.795,-64.413,394.736,165.232,58.558,160.389
C02577=1014.800,-64.163,394.725,165.235,58.551,160.388
C02578=1014.805,-63.914,394.716,165.238,58.544,160.388
C02579=1014.810,-63.664,394.706,165.240,58.537,160.387
C02580=1014.815,-63.414,394.696,165.243,58.530,160.387
C02581=1014.820,-63.164,394.687,165.246,58.523,160.386
C02582=1014.825,-62.915,394.677,165.248,58.516,160.385
C02583=1014.830,-62.665,394.667,165.250,58.509,160.385
C02584=1014.835,-62.415,394.657,165.254,58.503,160.384
C02585=1014.840,-62.166,394.647,165.257,58.496,160.384
C02586=1014.844,-61.915,394.637,165.259,58.488,160.383
C02587=1014.849,-61.665,394.627,165.262,58.481,160.383
C02588=1014.854,-61.416,394.617,165.265,58.474,160.382
C02589=1014.859,-61.166,394.607,165.268,58.467,160.382
C02590=1014.864,-60.916,394.598,165.270,58.459,160.381
C02591=1014.869,-60.667,394.588,165.272,58.452,160.380
C02592=1014.874,-60.417,394.578,165.275,58.445,160.380
C02593=1014.879,-60.168,394.568,165.278,58.438,160.379
C02594=1014.884,-59.917,394.558,165.281,58.431,160.378
C02595=1014.889,-59.668,394.548,165.284,58.424,160.378
C02596=1014.894,-59.418,394.539,165.286,58.417,160.377
C02597=1014.899,-59.168,394.529,165.289,58.409,160.377
C02598=1014.904,-58.918,394.519,165.292,58.402,160.376
C02599=1014.910,-58.668,394.509,165.295,58.395,160.376
C02600=1014.914,-58.419,394.499,165.297,58.388,160.375
C02601=1014.919,-58.170,394.489,165.299,58.380,160.374
C02602=1014.925,-57.919,394.479,165.302,58.373,160.374
C02603=1014.929,-57.670,394.469,165.305,58.366,160.373
C02604=1014.935,-57.420,394.459,165.308,58.359,160.372
C02605=1014.940,-57.170,394.449,165.311,58.352,160.372
C02606=1014.945,-56.920,394.439,165.313,58.345,160.371
C02607=1014.950,-56.671,394.429,165.315,58.337,160.370
C02608=1014.955,-56.421,394.419,165.318,58.330,160.370
C02609=1014.960,-56.171,394.409,165.321,58.323,160.369
C02610=1014.966,-55.921,394.399,165.324,58.316,160.369
C02611=1014.970,-55.672,394.389,165.326,58.308,160.368
C02612=1014.975,-55.422,394.378,165.329,58.301,160.367
C02613=1014.980,-55.172,394.369,165.332,58.294,160.367
C02614=1014.986,-54.922,394.359,165.334,58.287,160.366
C02615=1014.990,-54.673,394.349,165.336,58.279,160.365
C02616=1014.996,-54.422,394.339,165.339,58.272,160.365
C02617=1015.001,-54.148,394.328,165.343,58.263,160.364
C02618=1015.007,-53.872,394.316,165.346,58.255,160.363
C02619=1015.013,-53.596,394.306,165.348,58.247,160.362
C02620=1015.019,-53.320,394.294,165.351,58.239,160.362
C02621=1015.023,-53.070,394.284,165.354,58.232,160.361
C02622=1015.029,-52.820,394.274,165.356,58.224,160.360
C02623=1015.034,-52.570,394.264,165.360,58.217,160.360
C02624=1015.039,-52.321,394.254,165.362,58.209,160.359
C02625=1015.044,-52.070,394.244,165.365,58.202,160.358
C02626=1015.049,-51.821,394.234,165.368,58.195,160.358
C02627=1015.055,-51.572,394.223,165.370,58.187,160.357
C02628=1015.060,-51.322,394.213,165.373,58.180,160.356
C02629=1015.065,-51.072,394.203,165.375,58.172,160.355
C02630=1015.070,-50.822,394.192,165.378,58.165,160.355
C02631=1015.074,-50.573,394.181,165.381,58.158,160.354
C02632=1015.080,-50.322,394.171,165.383,58.151,160.354
C02633=1015.085,-50.072,394.160,165.386,58.144,160.353
C02634=1015.090,-49.823,394.150,165.389,58.137,160.353
C02635=1015.094,-49.573,394.139,165.391,58.129,160.352
C02636=1015.100,-49.324,394.129,165.394,58.122,160.351
C02637=1015.104,-49.074,394.118,165.397,58.115,160.351
C02638=1015.110,-48.823,394.108,165.400,58.108,160.350
C02639=1015.115,-48.575,394.097,165.402,58.100,160.349
C02640=1015.119,-48.324,394.086,165.405,58.093,160.349
C02641=1015.125,-48.075,394.075,165.407,58.086,160.348
C02642=1015.129,-47.825,394.065,165.410,58.079,160.347
C02643=1015.135,-47.576,394.054,165.412,58.071,160.347
C02644=1015.140,-47.325,394.043,165.415,58.064,160.346
C02645=1015.145,-47.076,394.033,165.418,58.057,160.345
C02646=1015.150,-46.826,394.022,165.421,58.050,160.345
C02647=1015.155,-46.576,394.012,165.423,58.042,160.344
C02648=1015.159,-46.327,394.001,165.426,58.035,160.343
C02649=1015.165,-46.077,393.991,165.429,58.028,160.343
C02650=1015.170,-45.827,393.979,165.431,58.020,160.342
C02651=1015.175,-45.578,393.969,165.434,58.013,160.341
C02652=1015.180,-45.328,393.958,165.436,58.005,160.340
C02653=1015.185,-45.078,393.947,165.439,57.998,160.340
C02654=1015.190,-44.828,393.937,165.443,57.990,160.340
C02655=1015.195,-44.579,393.926,165.445,57.983,160.339
C02656=1015.201,-44.329,393.916,165.448,57.976,160.338
C02657=1015.205,-44.080,393.905,165.450,57.968,160.337
C02658=1015.211,-43.830,393.894,165.453,57.961,160.337
C02659=1015.216,-43.580,393.883,165.456,57.954,160.336
C02660=1015.221,-43.330,393.873,165.458,57.946,160.335
C02661=1015.225,-43.081,393.862,165.461,57.939,160.335
C02662=1015.231,-42.831,393.851,165.463,57.931,160.334
C02663=1015.236,-42.581,393.840,165.466,57.924,160.333
C02664=1015.242,-42.331,393.829,165.469,57.916,160.332
C02665=1015.246,-42.081,393.819,165.472,57.909,160.332
C02666=1015.251,-41.832,393.808,165.474,57.901,160.331
C02667=1015.256,-41.582,393.796,165.477,57.894,160.330
C02668=1015.262,-41.332,393.786,165.479,57.886,160.330
C02669=1015.266,-41.083,393.775,165.482,57.879,160.329
C02670=1015.272,-40.833,393.764,165.484,57.871,160.328
C02671=1015.277,-40.583,393.754,165.487,57.864,160.328
C02672=1015.282,-40.334,393.743,165.490,57.856,160.327
C02673=1015.287,-40.083,393.732,165.493,57.848,160.326
C02674=1015.292,-39.834,393.721,165.495,57.841,160.325
C02675=1015.297,-39.585,393.710,165.498,57.833,160.325
C02676=1015.303,-39.335,393.699,165.500,57.826,160.324
C02677=1015.308,-39.085,393.688,165.503,57.819,160.323
C02678=1015.313,-38.835,393.677,165.506,57.812,160.323
C02679=1015.318,-38.585,393.665,165.508,57.805,160.322
C02680=1015.323,-38.336,393.655,165.511,57.797,160.321
C02681=1015.328,-38.061,393.642,165.514,57.789,160.320
C02682=1015.333,-37.785,393.630,165.517,57.780,160.320
C02683=1015.339,-37.510,393.618,165.520,57.773,160.319
C02684=1015.345,-37.234,393.606,165.523,57.764,160.318
C02685=1015.350,-36.984,393.594,165.525,57.757,160.317
C02686=1015.355,-36.734,393.583,165.528,57.750,160.317
C02687=1015.360,-36.484,393.571,165.530,57.742,160.316
C02688=1015.366,-36.235,393.561,165.534,57.734,160.315
C02689=1015.371,-35.985,393.549,165.536,57.727,160.315
C02690=1015.376,-35.735,393.538,165.539,57.719,160.314
C02691=1015.381,-35.485,393.526,165.542,57.712,160.313
C02692=1015.386,-35.237,393.516,165.544,57.704,160.312
C02693=1015.390,-34.986,393.505,165.547,57.697,160.312
C02694=1015.395,-34.736,393.493,165.549,57.689,160.311
C02695=1015.400,-34.487,393.482,165.552,57.682,160.310
C02696=1015.406,-34.237,393.471,165.554,57.675,160.309
C02697=1015.411,-33.987,393.460,165.557,57.666,160.309
C02698=1015.416,-33.737,393.448,165.560,57.659,160.308
C02699=1015.421,-33.488,393.437,165.563,57.652,160.307
C02700=1015.427,-33.238,393.426,165.565,57.645,160.307
C02701=1015.435,-32.836,393.407,165.570,57.632,160.305
C02702=1015.443,-32.432,393.390,165.574,57.620,160.304
C02703=1015.451,-32.029,393.371,165.578,57.607,160.303
C02704=1015.459,-31.626,393.352,165.582,57.595,160.302
C02705=1015.465,-31.376,393.341,165.585,57.588,160.301
C02706=1015.470,-31.127,393.330,165.587,57.580,160.300
C02707=1015.475,-30.877,393.318,165.590,57.572,160.299
C02708=1015.480,-30.627,393.307,165.593,57.565,160.299
C02709=1015.486,-30.377,393.296,165.596,57.557,160.298
C02710=1015.491,-30.128,393.284,165.598,57.549,160.297
C02711=1015.496,-29.878,393.273,165.601,57.542,160.296
C02712=1015.501,-29.628,393.261,165.603,57.534,160.296
C02713=1015.507,-29.379,393.251,165.607,57.527,160.295
C02714=1015.512,-29.129,393.239,165.609,57.519,160.294
C02715=1015.517,-28.880,393.227,165.611,57.511,160.293
C02716=1015.522,-28.630,393.215,165.614,57.503,160.293
C02717=1015.527,-28.380,393.204,165.616,57.496,160.292
C02718=1015.533,-28.130,393.193,165.620,57.488,160.291
C02719=1015.538,-27.881,393.182,165.622,57.480,160.290
C02720=1015.543,-27.631,393.170,165.625,57.473,160.290
C02721=1015.548,-27.381,393.159,165.627,57.465,160.289
C02722=1015.553,-27.132,393.146,165.630,57.458,160.288
C02723=1015.558,-26.882,393.135,165.632,57.450,160.287
C02724=1015.563,-26.632,393.124,165.634,57.443,160.286
C02725=1015.568,-26.383,393.111,165.638,57.435,160.286
C02726=1015.572,-26.133,393.099,165.641,57.427,160.285
C02727=1015.578,-25.882,393.087,165.643,57.420,160.284
C02728=1015.583,-25.633,393.075,165.646,57.413,160.284
C02729=1015.588,-25.384,393.064,165.648,57.405,160.283
C02730=1015.593,-25.134,393.052,165.650,57.397,160.282
C02731=1015.599,-24.885,393.040,165.653,57.390,160.281
C02732=1015.604,-24.635,393.029,165.656,57.383,160.281
C02733=1015.609,-24.385,393.017,165.659,57.374,160.280
C02734=1015.614,-24.136,393.005,165.661,57.367,160.279
C02735=1015.619,-23.886,392.994,165.664,57.359,160.278
C02736=1015.624,-23.636,392.982,165.667,57.352,160.278
C02737=1015.629,-23.387,392.970,165.669,57.344,160.277
C02738=1015.635,-23.136,392.958,165.671,57.337,160.276
C02739=1015.640,-22.887,392.947,165.675,57.328,160.275
C02740=1015.645,-22.637,392.934,165.677,57.321,160.274
C02741=1015.652,-22.265,392.917,165.681,57.310,160.273
C02742=1015.660,-21.891,392.899,165.685,57.298,160.272
C02743=1015.668,-21.519,392.881,165.689,57.287,160.271
C02744=1015.675,-21.146,392.863,165.693,57.275,160.270
C02745=1015.681,-20.896,392.851,165.696,57.268,160.269
C02746=1015.686,-20.647,392.840,165.698,57.260,160.268
C02747=1015.691,-20.397,392.828,165.700,57.252,160.267
C02748=1015.697,-20.147,392.816,165.704,57.244,160.267
C02749=1015.702,-19.897,392.804,165.706,57.237,160.266
C02750=1015.707,-19.648,392.792,165.708,57.229,160.265
C02751=1015.712,-19.398,392.780,165.711,57.221,160.264
C02752=1015.717,-19.149,392.768,165.714,57.213,160.263
C02753=1015.723,-18.898,392.756,165.717,57.205,160.263
C02754=1015.728,-18.649,392.744,165.719,57.198,160.262
C02755=1015.732,-18.399,392.732,165.721,57.190,160.261
C02756=1015.738,-18.150,392.720,165.725,57.182,160.260
C02757=1015.743,-17.900,392.709,165.727,57.174,160.259
C02758=1015.749,-17.650,392.696,165.729,57.166,160.258
C02759=1015.754,-17.400,392.684,165.732,57.159,160.258
C02760=1015.759,-17.151,392.672,165.735,57.151,160.257
C02761=1015.764,-16.902,392.661,165.738,57.143,160.256
C02762=1015.770,-16.652,392.648,165.740,57.135,160.255
C02763=1015.775,-16.402,392.636,165.742,57.128,160.254
C02764=1015.780,-16.153,392.625,165.746,57.119,160.254
C02765=1015.785,-15.903,392.612,165.748,57.112,160.253
C02766=1015.790,-15.653,392.600,165.750,57.104,160.252
C02767=1015.796,-15.403,392.588,165.753,57.096,160.251
C02768=1015.800,-15.154,392.575,165.755,57.089,160.250
C02769=1015.806,-14.904,392.562,165.758,57.081,160.249
C02770=1015.811,-14.654,392.551,165.762,57.074,160.249
C02771=1015.816,-14.405,392.538,165.764,57.066,160.248
C02772=1015.822,-14.155,392.526,165.766,57.058,160.247
C02773=1015.826,-13.905,392.514,165.769,57.051,160.246
C02774=1015.831,-13.656,392.501,165.771,57.043,160.245
C02775=1015.836,-13.406,392.489,165.774,57.035,160.245
C02776=1015.842,-13.156,392.476,165.777,57.027,160.244
C02777=1015.847,-12.907,392.464,165.779,57.019,160.243
C02778=1015.852,-12.657,392.452,165.782,57.012,160.242
C02779=1015.857,-12.407,392.439,165.784,57.004,160.241
C02780=1015.862,-12.158,392.427,165.786,56.996,160.241
C02781=1015.868,-11.909,392.415,165.790,56.988,160.240
C02782=1015.873,-11.658,392.402,165.792,56.981,160.239
C02783=1015.878,-11.409,392.390,165.795,56.973,160.238
C02784=1015.883,-11.160,392.378,165.797,56.965,160.237
C02785=1015.888,-10.909,392.365,165.800,56.957,160.237
C02786=1015.894,-10.660,392.353,165.803,56.950,160.236
C02787=1015.898,-10.411,392.340,165.805,56.942,160.235
C02788=1015.904,-10.161,392.327,165.808,56.934,160.234
C02789=1015.909,-9.911,392.316,165.810,56.927,160.233
C02790=1015.914,-9.661,392.303,165.814,56.919,160.233
C02791=1015.920,-9.412,392.291,165.816,56.911,160.232
C02792=1015.925,-9.162,392.278,165.818,56.902,160.231
C02793=1015.930,-8.912,392.265,165.820,56.895,160.230
C02794=1015.935,-8.663,392.253,165.824,56.887,160.229
C02795=1015.940,-8.414,392.240,165.826,56.879,160.228
C02796=1015.946,-8.164,392.228,165.828,56.871,160.227
C02797=1015.951,-7.914,392.216,165.831,56.864,160.226
C02798=1015.956,-7.664,392.203,165.834,56.856,160.226
C02799=1015.961,-7.414,392.191,165.837,56.848,160.225
C02800=1015.967,-7.165,392.179,165.839,56.840,160.224
C02801=1015.972,-6.915,392.166,165.842,56.832,160.223
C02802=1015.977,-6.666,392.153,165.844,56.824,160.222
C02803=1015.983,-6.416,392.141,165.847,56.816,160.221
C02804=1015.988,-6.167,392.128,165.849,56.809,160.221
C02805=1015.993,-5.888,392.114,165.852,56.800,160.220
C02806=1015.999,-5.609,392.100,165.855,56.790,160.218
C02807=1016.006,-5.331,392.087,165.857,56.781,160.217
C02808=1016.012,-5.054,392.072,165.860,56.773,160.216
C02809=1016.017,-4.803,392.059,165.864,56.765,160.216
C02810=1016.022,-4.554,392.047,165.866,56.757,160.215
C02811=1016.027,-4.304,392.034,165.869,56.749,160.214
C02812=1016.032,-4.055,392.021,165.871,56.742,160.213
C02813=1016.038,-3.805,392.008,165.875,56.734,160.213
C02814=1016.042,-3.555,391.996,165.877,56.726,160.212
C02815=1016.047,-3.305,391.982,165.880,56.718,160.211
C02816=1016.053,-3.056,391.969,165.882,56.711,160.210
C02817=1016.058,-2.806,391.956,165.884,56.703,160.209
C02818=1016.063,-2.557,391.944,165.887,56.695,160.208
C02819=1016.068,-2.306,391.930,165.889,56.688,160.207
C02820=1016.073,-2.057,391.918,165.892,56.679,160.206
C02821=1016.079,-1.808,391.904,165.895,56.671,160.206
C02822=1016.083,-1.558,391.892,165.897,56.664,160.205
C02823=1016.088,-1.308,391.878,165.900,56.656,160.204
C02824=1016.094,-1.059,391.866,165.902,56.649,160.203
C02825=1016.099,-0.809,391.852,165.904,56.641,160.202
C02826=1016.104,-0.560,391.840,165.908,56.633,160.202
C02827=1016.109,-0.310,391.826,165.910,56.625,160.201
C02828=1016.115,-0.061,391.814,165.913,56.618,160.200
C02829=1016.120,0.189,391.800,165.915,56.610,160.199
C02830=1016.124,0.439,391.788,165.917,56.602,160.198
C02831=1016.130,0.688,391.774,165.920,56.594,160.197
C02832=1016.135,0.937,391.762,165.923,56.586,160.196
C02833=1016.140,1.188,391.748,165.926,56.578,160.196
C02834=1016.145,1.438,391.735,165.928,56.571,160.195
C02835=1016.150,1.687,391.722,165.931,56.563,160.194
C02836=1016.156,1.937,391.709,165.932,56.555,160.193
C02837=1016.161,2.186,391.696,165.936,56.547,160.192
C02838=1016.166,2.436,391.683,165.938,56.539,160.191
C02839=1016.171,2.685,391.670,165.941,56.532,160.190
C02840=1016.177,2.934,391.657,165.943,56.524,160.189
C02841=1016.182,3.185,391.643,165.946,56.515,160.189
C02842=1016.187,3.434,391.631,165.949,56.508,160.188
C02843=1016.192,3.684,391.617,165.951,56.500,160.187
C02844=1016.198,3.933,391.605,165.954,56.492,160.186
C02845=1016.203,4.183,391.591,165.957,56.484,160.185
C02846=1016.208,4.433,391.578,165.959,56.476,160.184
C02847=1016.213,4.682,391.565,165.962,56.468,160.183
C02848=1016.219,4.931,391.551,165.964,56.460,160.182
C02849=1016.224,5.181,391.539,165.967,56.452,160.182
C02850=1016.229,5.431,391.526,165.970,56.444,160.181
C02851=1016.234,5.681,391.512,165.972,56.436,160.180
C02852=1016.239,5.930,391.499,165.974,56.428,160.179
C02853=1016.245,6.179,391.486,165.978,56.420,160.178
C02854=1016.250,6.430,391.472,165.980,56.412,160.177
C02855=1016.255,6.678,391.459,165.982,56.405,160.176
C02856=1016.260,6.929,391.446,165.984,56.397,160.175
C02857=1016.266,7.178,391.433,165.987,56.388,160.174
C02858=1016.271,7.427,391.420,165.990,56.381,160.173
C02859=1016.276,7.677,391.406,165.992,56.373,160.173
C02860=1016.282,7.927,391.393,165.995,56.364,160.172
C02861=1016.287,8.176,391.381,165.998,56.357,160.171
C02862=1016.292,8.426,391.367,166.000,56.348,160.170
C02863=1016.298,8.676,391.354,166.002,56.341,160.169
C02864=1016.302,8.925,391.340,166.006,56.333,160.168
C02865=1016.308,9.175,391.328,166.008,56.324,160.167
C02866=1016.314,9.424,391.314,166.010,56.317,160.166
C02867=1016.319,9.673,391.300,166.013,56.308,160.165
C02868=1016.324,9.924,391.287,166.016,56.301,160.164
C02869=1016.330,10.204,391.272,166.018,56.291,160.163
C02870=1016.336,10.484,391.257,166.021,56.282,160.162
C02871=1016.342,10.765,391.242,166.024,56.274,160.161
C02872=1016.348,11.046,391.227,166.027,56.264,160.160
C02873=1016.353,11.295,391.213,166.030,56.256,160.159
C02874=1016.359,11.544,391.201,166.032,56.248,160.158
C02875=1016.364,11.794,391.187,166.035,56.240,160.157
C02876=1016.369,12.044,391.174,166.038,56.232,160.157
C02877=1016.375,12.294,391.160,166.040,56.224,160.156
C02878=1016.381,12.542,391.147,166.042,56.216,160.155
C02879=1016.386,12.793,391.134,166.046,56.207,160.154
C02880=1016.391,13.042,391.120,166.048,56.199,160.153
C02881=1016.397,13.292,391.107,166.050,56.191,160.152
C02882=1016.402,13.542,391.093,166.054,56.183,160.151
C02883=1016.407,13.791,391.080,166.056,56.176,160.150
C02884=1016.412,14.040,391.066,166.058,56.167,160.149
C02885=1016.417,14.291,391.053,166.061,56.160,160.148
C02886=1016.423,14.540,391.039,166.063,56.152,160.147
C02887=1016.428,14.790,391.025,166.066,56.143,160.146
C02888=1016.432,15.039,391.011,166.069,56.136,160.146
C02889=1016.438,15.288,390.997,166.071,56.128,160.144
C02890=1016.443,15.539,390.984,166.073,56.120,160.144
C02891=1016.449,15.788,390.970,166.077,56.112,160.143
C02892=1016.454,16.038,390.956,166.079,56.104,160.142
C02893=1016.459,16.287,390.943,166.081,56.096,160.141
C02894=1016.464,16.536,390.929,166.083,56.088,160.140
C02895=1016.470,16.786,390.916,166.087,56.080,160.139
C02896=1016.475,17.036,390.902,166.089,56.072,160.138
C02897=1016.480,17.286,390.888,166.092,56.064,160.137
C02898=1016.485,17.534,390.875,166.094,56.056,160.136
C02899=1016.491,17.784,390.861,166.097,56.048,160.136
C02900=1016.496,18.034,390.847,166.099,56.040,160.134
C02901=1016.502,18.283,390.833,166.102,56.032,160.134
C02902=1016.507,18.533,390.819,166.104,56.024,160.132
C02903=1016.512,18.783,390.805,166.107,56.016,160.132
C02904=1016.517,19.032,390.792,166.109,56.008,160.131
C02905=1016.522,19.282,390.778,166.112,56.000,160.130
C02906=1016.528,19.531,390.764,166.114,55.992,160.129
C02907=1016.533,19.781,390.750,166.118,55.984,160.128
C02908=1016.538,20.031,390.736,166.120,55.976,160.127
C02909=1016.543,20.280,390.722,166.122,55.968,160.126
C02910=1016.549,20.530,390.708,166.125,55.960,160.125
C02911=1016.554,20.779,390.694,166.128,55.952,160.124
C02912=1016.559,21.028,390.681,166.130,55.944,160.124
C02913=1016.564,21.278,390.666,166.132,55.936,160.122
C02914=1016.569,21.528,390.652,166.135,55.928,160.122
C02915=1016.575,21.777,390.639,166.137,55.920,160.120
C02916=1016.580,22.027,390.625,166.141,55.912,160.120
C02917=1016.585,22.277,390.610,166.143,55.904,160.119
C02918=1016.590,22.526,390.596,166.145,55.896,160.118
C02919=1016.596,22.776,390.583,166.147,55.888,160.117
C02920=1016.601,23.026,390.569,166.151,55.880,160.116
C02921=1016.607,23.274,390.554,166.153,55.872,160.115
C02922=1016.611,23.524,390.540,166.155,55.864,160.114
C02923=1016.617,23.773,390.526,166.157,55.856,160.113
C02924=1016.622,24.023,390.512,166.161,55.848,160.112
C02925=1016.628,24.272,390.498,166.163,55.840,160.111
C02926=1016.632,24.522,390.484,166.165,55.832,160.110
C02927=1016.638,24.772,390.470,166.169,55.824,160.109
C02928=1016.643,25.021,390.456,166.171,55.816,160.108
C02929=1016.649,25.271,390.442,166.174,55.808,160.108
C02930=1016.654,25.521,390.428,166.176,55.800,160.106
C02931=1016.659,25.770,390.413,166.179,55.791,160.106
C02932=1016.665,26.019,390.399,166.181,55.784,160.105
C02933=1016.671,26.301,390.384,166.184,55.774,160.103
C02934=1016.677,26.584,390.368,166.187,55.766,160.103
C02935=1016.682,26.865,390.351,166.190,55.756,160.101
C02936=1016.689,27.148,390.335,166.192,55.747,160.100
C02937=1016.693,27.397,390.322,166.196,55.739,160.099
C02938=1016.700,27.647,390.307,166.198,55.731,160.098
C02939=1016.705,27.896,390.292,166.200,55.723,160.098
C02940=1016.710,28.146,390.279,166.203,55.715,160.096
C02941=1016.715,28.396,390.264,166.205,55.707,160.096
C02942=1016.721,28.645,390.250,166.207,55.699,160.095
C02943=1016.725,28.895,390.235,166.211,55.691,160.094
C02944=1016.731,29.144,390.221,166.213,55.683,160.093
C02945=1016.736,29.394,390.206,166.216,55.676,160.092
C02946=1016.741,29.643,390.192,166.218,55.667,160.091
C02947=1016.746,29.893,390.178,166.221,55.659,160.090
C02948=1016.752,30.142,390.163,166.223,55.651,160.089
C02949=1016.757,30.392,390.149,166.226,55.643,160.088
C02950=1016.762,30.641,390.135,166.228,55.636,160.087
C02951=1016.767,30.891,390.120,166.230,55.627,160.086
C02952=1016.773,31.140,390.106,166.234,55.619,160.085
C02953=1016.777,31.390,390.091,166.236,55.611,160.084
C02954=1016.783,31.639,390.077,166.239,55.604,160.083
C02955=1016.788,31.889,390.062,166.241,55.595,160.082
C02956=1016.794,32.138,390.048,166.244,55.587,160.081
C02957=1016.798,32.388,390.033,166.246,55.579,160.081
C02958=1016.804,32.637,390.019,166.249,55.571,160.079
C02959=1016.809,32.887,390.004,166.251,55.563,160.078
C02960=1016.814,33.136,389.990,166.254,55.555,160.078
C02961=1016.820,33.385,389.976,166.256,55.547,160.077
C02962=1016.825,33.635,389.961,166.259,55.539,160.076
C02963=1016.830,33.885,389.947,166.261,55.531,160.075
C02964=1016.836,34.135,389.932,166.264,55.523,160.074
C02965=1016.841,34.384,389.918,166.266,55.514,160.073
C02966=1016.846,34.634,389.903,166.269,55.507,160.072
C02967=1016.852,34.883,389.889,166.272,55.498,160.071
C02968=1016.857,35.132,389.874,166.274,55.490,160.070
C02969=1016.862,35.382,389.860,166.277,55.483,160.069
C02970=1016.868,35.631,389.845,166.279,55.474,160.068
C02971=1016.873,35.881,389.831,166.282,55.466,160.067
C02972=1016.878,36.130,389.816,166.284,55.458,160.066
C02973=1016.884,36.380,389.801,166.287,55.450,160.065
C02974=1016.889,36.630,389.786,166.289,55.442,160.064
C02975=1016.894,36.879,389.772,166.292,55.433,160.063
C02976=1016.899,37.129,389.757,166.295,55.426,160.062
C02977=1016.904,37.378,389.743,166.297,55.418,160.061
C02978=1016.909,37.628,389.728,166.300,55.410,160.060
C02979=1016.914,37.877,389.712,166.302,55.402,160.059
C02980=1016.920,38.127,389.698,166.305,55.393,160.058
C02981=1016.926,38.376,389.683,166.308,55.386,160.057
C02982=1016.931,38.626,389.668,166.310,55.378,160.056
C02983=1016.935,38.876,389.653,166.313,55.370,160.056
C02984=1016.941,39.124,389.639,166.315,55.362,160.054
C02985=1016.946,39.374,389.624,166.318,55.353,160.054
C02986=1016.952,39.624,389.609,166.321,55.346,160.053
C02987=1016.957,39.874,389.594,166.323,55.338,160.052
C02988=1016.962,40.123,389.579,166.325,55.330,160.051
C02989=1016.967,40.372,389.565,166.328,55.322,160.050
C02990=1016.972,40.622,389.549,166.331,55.314,160.049
C02991=1016.977,40.871,389.534,166.333,55.305,160.048
C02992=1016.983,41.121,389.520,166.336,55.298,160.047
C02993=1016.988,41.371,389.505,166.338,55.290,160.046
C02994=1016.993,41.620,389.490,166.341,55.281,160.045
C02995=1016.998,41.869,389.475,166.344,55.274,160.044
C02996=1017.004,42.119,389.461,166.346,55.266,160.043
C02997=1017.010,42.401,389.443,166.349,55.256,160.042
C02998=1017.015,42.683,389.426,166.352,55.248,160.041
C02999=1017.022,42.965,389.408,166.355,55.238,160.040
C03000=1017.028,43.247,389.391,166.358,55.230,160.039
C03001=1017.033,43.496,389.376,166.360,55.222,160.038
C03002=1017.038,43.746,389.362,166.363,55.214,160.037
C03003=1017.043,43.996,389.346,166.365,55.206,160.036
C03004=1017.048,44.245,389.331,166.367,55.198,160.035
C03005=1017.053,44.495,389.316,166.370,55.190,160.034
C03006=1017.058,44.744,389.300,166.373,55.182,160.033
C03007=1017.063,44.993,389.285,166.376,55.174,160.032
C03008=1017.068,45.243,389.269,166.378,55.166,160.031
C03009=1017.073,45.493,389.254,166.380,55.159,160.030
C03010=1017.078,45.742,389.239,166.383,55.151,160.029
C03011=1017.083,45.991,389.224,166.385,55.143,160.028
C03012=1017.088,46.241,389.208,166.388,55.135,160.027
C03013=1017.094,46.491,389.193,166.391,55.127,160.026
C03014=1017.099,46.740,389.178,166.393,55.118,160.025
C03015=1017.104,46.989,389.163,166.396,55.111,160.024
C03016=1017.109,47.238,389.147,166.398,55.103,160.023
C03017=1017.115,47.488,389.132,166.400,55.095,160.022
C03018=1017.120,47.738,389.117,166.403,55.087,160.021
C03019=1017.125,47.987,389.101,166.406,55.079,160.020
C03020=1017.131,48.237,389.086,166.409,55.071,160.020
C03021=1017.136,48.486,389.071,166.411,55.063,160.019
C03022=1017.141,48.735,389.056,166.413,55.055,160.018
C03023=1017.146,48.985,389.040,166.415,55.047,160.016
C03024=1017.151,49.235,389.025,166.418,55.039,160.016
C03025=1017.156,49.484,389.010,166.421,55.031,160.015
C03026=1017.161,49.733,388.995,166.424,55.023,160.014
C03027=1017.167,49.983,388.979,166.426,55.015,160.013
C03028=1017.172,50.232,388.964,166.428,55.007,160.012
C03029=1017.177,50.482,388.949,166.431,54.999,160.011
C03030=1017.183,50.732,388.933,166.434,54.991,160.010
C03031=1017.188,50.981,388.918,166.437,54.983,160.009
C03032=1017.193,51.230,388.901,166.439,54.975,160.008
C03033=1017.198,51.480,388.886,166.441,54.967,160.007
C03034=1017.203,51.729,388.871,166.444,54.958,160.006
C03035=1017.208,51.978,388.856,166.447,54.951,160.005
C03036=1017.214,52.228,388.840,166.449,54.943,160.004
C03037=1017.219,52.478,388.825,166.452,54.935,160.003
C03038=1017.224,52.727,388.810,166.454,54.927,160.002
C03039=1017.230,52.977,388.794,166.457,54.918,160.001
C03040=1017.235,53.226,388.779,166.460,54.911,160.000
C03041=1017.241,53.475,388.763,166.462,54.903,159.999
C03042=1017.246,53.725,388.748,166.464,54.894,159.998
C03043=1017.251,53.974,388.732,166.468,54.886,159.997
C03044=1017.256,54.224,388.717,166.470,54.878,159.996
C03045=1017.261,54.473,388.702,166.473,54.870,159.995
C03046=1017.267,54.723,388.686,166.475,54.862,159.994
C03047=1017.272,54.972,388.671,166.478,54.854,159.993
C03048=1017.277,55.221,388.655,166.480,54.846,159.992
C03049=1017.283,55.471,388.639,166.483,54.838,159.991
C03050=1017.288,55.720,388.624,166.485,54.829,159.990
C03051=1017.293,55.971,388.608,166.488,54.821,159.989
C03052=1017.298,56.220,388.593,166.491,54.814,159.988
C03053=1017.303,56.469,388.577,166.493,54.805,159.987
C03054=1017.309,56.719,388.562,166.495,54.797,159.986
C03055=1017.314,56.968,388.546,166.499,54.789,159.985
C03056=1017.320,57.218,388.531,166.501,54.781,159.984
C03057=1017.325,57.467,388.516,166.503,54.773,159.983
C03058=1017.331,57.716,388.499,166.505,54.764,159.982
C03059=1017.336,57.966,388.484,166.509,54.756,159.981
C03060=1017.341,58.216,388.469,166.511,54.748,159.980
C03061=1017.347,58.497,388.451,166.514,54.739,159.979
C03062=1017.353,58.779,388.434,166.517,54.729,159.978
C03063=1017.360,59.061,388.416,166.519,54.720,159.976
C03064=1017.366,59.343,388.398,166.522,54.711,159.975
C03065=1017.371,59.593,388.383,166.526,54.703,159.974
C03066=1017.377,59.842,388.367,166.528,54.694,159.973
C03067=1017.382,60.091,388.352,166.531,54.687,159.972
C03068=1017.387,60.341,388.336,166.534,54.679,159.972
C03069=1017.393,60.590,388.320,166.536,54.671,159.970
C03070=1017.398,60.840,388.304,166.539,54.662,159.969
C03071=1017.403,61.089,388.289,166.542,54.654,159.968
C03072=1017.409,61.339,388.273,166.544,54.646,159.967
C03073=1017.414,61.588,388.258,166.546,54.638,159.966
C03074=1017.419,61.838,388.242,166.550,54.629,159.965
C03075=1017.424,62.087,388.227,166.552,54.621,159.964
C03076=1017.430,62.337,388.211,166.554,54.613,159.963
C03077=1017.435,62.586,388.196,166.557,54.604,159.962
C03078=1017.441,62.835,388.179,166.560,54.597,159.961
C03079=1017.446,63.085,388.163,166.562,54.589,159.960
C03080=1017.451,63.335,388.148,166.565,54.580,159.959
C03081=1017.457,63.583,388.132,166.567,54.572,159.958
C03082=1017.461,63.834,388.116,166.570,54.564,159.957
C03083=1017.467,64.082,388.100,166.573,54.556,159.956
C03084=1017.472,64.332,388.083,166.575,54.548,159.955
C03085=1017.478,64.582,388.068,166.578,54.540,159.954
C03086=1017.483,64.831,388.052,166.581,54.532,159.953
C03087=1017.488,65.081,388.036,166.583,54.524,159.952
C03088=1017.493,65.330,388.020,166.586,54.516,159.951
C03089=1017.499,65.580,388.004,166.588,54.508,159.950
C03090=1017.504,65.829,387.988,166.590,54.500,159.949
C03091=1017.509,66.079,387.972,166.594,54.491,159.948
C03092=1017.514,66.327,387.956,166.596,54.484,159.947
C03093=1017.520,66.577,387.939,166.599,54.476,159.946
C03094=1017.525,66.827,387.923,166.601,54.468,159.945
C03095=1017.530,67.076,387.907,166.604,54.459,159.944
C03096=1017.536,67.326,387.892,166.607,54.451,159.943
C03097=1017.540,67.575,387.875,166.609,54.443,159.942
C03098=1017.546,67.824,387.859,166.611,54.435,159.941
C03099=1017.551,68.074,387.843,166.614,54.427,159.940
C03100=1017.556,68.323,387.827,166.618,54.419,159.939
C03101=1017.562,68.573,387.810,166.620,54.411,159.938
C03102=1017.567,68.822,387.795,166.622,54.403,159.937
C03103=1017.572,69.072,387.778,166.625,54.395,159.936
C03104=1017.577,69.321,387.761,166.627,54.387,159.935
C03105=1017.582,69.570,387.745,166.630,54.379,159.934
C03106=1017.587,69.820,387.729,166.633,54.371,159.934
C03107=1017.593,70.069,387.713,166.635,54.363,159.932
C03108=1017.598,70.318,387.697,166.638,54.355,159.931
C03109=1017.604,70.568,387.680,166.640,54.347,159.930
C03110=1017.608,70.817,387.665,166.644,54.339,159.929
C03111=1017.613,71.067,387.648,166.646,54.331,159.928
C03112=1017.619,71.316,387.631,166.648,54.323,159.927
C03113=1017.624,71.565,387.615,166.651,54.315,159.926
C03114=1017.629,71.815,387.598,166.653,54.307,159.925
C03115=1017.634,72.064,387.583,166.657,54.299,159.925
C03116=1017.639,72.314,387.566,166.659,54.291,159.923
C03117=1017.645,72.563,387.550,166.662,54.283,159.922
C03118=1017.650,72.812,387.533,166.664,54.275,159.921
C03119=1017.655,73.062,387.517,166.666,54.267,159.920
C03120=1017.661,73.311,387.500,166.670,54.258,159.919
C03121=1017.665,73.561,387.484,166.672,54.250,159.918
C03122=1017.671,73.810,387.468,166.675,54.243,159.918
C03123=1017.677,74.060,387.451,166.677,54.235,159.916
C03124=1017.681,74.309,387.435,166.680,54.227,159.915
C03125=1017.688,74.591,387.417,166.684,54.217,159.914
C03126=1017.693,74.873,387.398,166.687,54.208,159.913
C03127=1017.700,75.155,387.379,166.689,54.199,159.912
C03128=1017.706,75.437,387.361,166.692,54.190,159.911
C03129=1017.711,75.686,387.344,166.695,54.182,159.910
C03130=1017.716,75.935,387.327,166.697,54.174,159.909
C03131=1017.721,76.185,387.310,166.700,54.166,159.908
C03132=1017.726,76.434,387.295,166.703,54.158,159.907
C03133=1017.731,76.684,387.278,166.705,54.150,159.906
C03134=1017.737,76.934,387.262,166.708,54.142,159.905
C03135=1017.742,77.183,387.245,166.710,54.134,159.904
C03136=1017.747,77.432,387.229,166.713,54.126,159.903
C03137=1017.753,77.681,387.211,166.715,54.118,159.902
C03138=1017.758,77.931,387.194,166.719,54.110,159.901
C03139=1017.763,78.180,387.178,166.721,54.102,159.900
C03140=1017.768,78.429,387.161,166.724,54.094,159.899
C03141=1017.773,78.679,387.144,166.726,54.087,159.898
C03142=1017.778,78.929,387.127,166.729,54.079,159.897
C03143=1017.783,79.178,387.111,166.731,54.071,159.896
C03144=1017.788,79.427,387.094,166.735,54.062,159.895
C03145=1017.793,79.677,387.077,166.737,54.054,159.894
C03146=1017.798,79.927,387.060,166.739,54.046,159.893
C03147=1017.804,80.175,387.044,166.742,54.039,159.892
C03148=1017.809,80.424,387.027,166.745,54.031,159.891
C03149=1017.814,80.674,387.010,166.747,54.023,159.890
C03150=1017.820,80.924,386.993,166.751,54.015,159.889
C03151=1017.824,81.172,386.977,166.753,54.007,159.888
C03152=1017.830,81.422,386.960,166.755,53.999,159.887
C03153=1017.835,81.671,386.942,166.758,53.991,159.886
C03154=1017.840,81.921,386.925,166.760,53.983,159.885
C03155=1017.845,82.170,386.909,166.764,53.974,159.884
C03156=1017.850,82.419,386.892,166.767,53.967,159.883
C03157=1017.855,82.669,386.875,166.769,53.959,159.882
C03158=1017.861,82.919,386.858,166.771,53.951,159.881
C03159=1017.867,83.167,386.841,166.774,53.943,159.880
C03160=1017.872,83.417,386.825,166.777,53.935,159.879
C03161=1017.877,83.666,386.808,166.780,53.927,159.878
C03162=1017.882,83.916,386.791,166.782,53.919,159.877
C03163=1017.887,84.165,386.774,166.785,53.911,159.876
C03164=1017.893,84.414,386.757,166.787,53.903,159.875
C03165=1017.898,84.664,386.740,166.791,53.894,159.874
C03166=1017.903,84.914,386.723,166.793,53.886,159.873
C03167=1017.908,85.163,386.707,166.795,53.878,159.872
C03168=1017.913,85.412,386.689,166.798,53.870,159.871
C03169=1017.918,85.661,386.672,166.801,53.862,159.870
C03170=1017.924,85.911,386.655,166.804,53.854,159.869
C03171=1017.929,86.161,386.638,166.806,53.846,159.868
C03172=1017.934,86.410,386.621,166.809,53.838,159.867
C03173=1017.940,86.658,386.605,166.812,53.830,159.866
C03174=1017.945,86.908,386.588,166.815,53.822,159.865
C03175=1017.950,87.157,386.571,166.817,53.814,159.864
C03176=1017.956,87.407,386.554,166.819,53.806,159.863
C03177=1017.961,87.656,386.537,166.823,53.797,159.862
C03178=1017.966,87.906,386.519,166.825,53.789,159.861
C03179=1017.971,88.155,386.502,166.828,53.782,159.860
C03180=1017.977,88.405,386.486,166.830,53.774,159.859
C03181=1017.982,88.655,386.469,166.834,53.765,159.858
C03182=1017.987,88.903,386.452,166.836,53.757,159.857
C03183=1017.992,89.152,386.435,166.839,53.749,159.856
C03184=1017.998,89.402,386.417,166.842,53.742,159.855
C03185=1018.002,89.652,386.400,166.844,53.734,159.854
C03186=1018.008,89.901,386.382,166.848,53.726,159.853
C03187=1018.013,90.150,386.365,166.850,53.718,159.852
C03188=1018.018,90.399,386.348,166.853,53.710,159.851
C03189=1018.023,90.681,386.328,166.856,53.701,159.850
C03190=1018.030,90.964,386.309,166.859,53.692,159.849
C03191=1018.035,91.246,386.289,166.862,53.683,159.848
C03192=1018.041,91.527,386.270,166.865,53.674,159.847
C03193=1018.046,91.776,386.252,166.868,53.666,159.846
C03194=1018.052,92.026,386.235,166.870,53.659,159.845
C03195=1018.056,92.275,386.217,166.873,53.651,159.844
C03196=1018.062,92.525,386.200,166.876,53.642,159.843
C03197=1018.067,92.774,386.183,166.879,53.634,159.842
C03198=1018.072,93.024,386.166,166.881,53.626,159.841
C03199=1018.077,93.273,386.148,166.884,53.618,159.840
C03200=1018.083,93.522,386.130,166.886,53.611,159.839
C03201=1018.088,93.772,386.113,166.890,53.602,159.838
C03202=1018.093,94.021,386.096,166.893,53.595,159.837
C03203=1018.098,94.271,386.078,166.895,53.587,159.836
C03204=1018.103,94.520,386.061,166.898,53.579,159.835
C03205=1018.109,94.769,386.043,166.900,53.571,159.834
C03206=1018.114,95.018,386.026,166.904,53.563,159.833
C03207=1018.119,95.268,386.008,166.906,53.555,159.832
C03208=1018.124,95.517,385.990,166.909,53.547,159.831
C03209=1018.130,95.767,385.974,166.911,53.539,159.830
C03210=1018.135,96.016,385.956,166.915,53.531,159.829
C03211=1018.140,96.266,385.939,166.917,53.523,159.828
C03212=1018.145,96.515,385.921,166.920,53.515,159.827
C03213=1018.151,96.764,385.903,166.922,53.507,159.826
C03214=1018.156,97.013,385.887,166.926,53.499,159.825
C03215=1018.161,97.263,385.868,166.928,53.491,159.824
C03216=1018.166,97.512,385.851,166.931,53.483,159.823
C03217=1018.172,97.761,385.833,166.933,53.475,159.822
C03218=1018.177,98.010,385.816,166.937,53.467,159.821
C03219=1018.182,98.260,385.798,166.939,53.459,159.820
C03220=1018.187,98.509,385.781,166.942,53.451,159.819
C03221=1018.192,98.758,385.764,166.944,53.443,159.818
C03222=1018.198,99.007,385.746,166.948,53.435,159.817
C03223=1018.203,99.257,385.728,166.950,53.427,159.816
C03224=1018.208,99.506,385.711,166.953,53.419,159.815
C03225=1018.213,99.756,385.693,166.955,53.411,159.814
C03226=1018.217,100.005,385.675,166.958,53.403,159.813
C03227=1018.223,100.254,385.657,166.961,53.396,159.812
C03228=1018.228,100.504,385.639,166.964,53.387,159.811
C03229=1018.233,100.753,385.622,166.967,53.380,159.810
C03230=1018.238,101.002,385.603,166.970,53.372,159.809
C03231=1018.243,101.251,385.586,166.972,53.364,159.808
C03232=1018.248,101.500,385.568,166.975,53.356,159.807
C03233=1018.254,101.749,385.550,166.978,53.348,159.806
C03234=1018.259,101.999,385.532,166.981,53.340,159.805
C03235=1018.264,102.249,385.514,166.984,53.333,159.804
C03236=1018.269,102.498,385.497,166.986,53.325,159.803
C03237=1018.274,102.748,385.478,166.989,53.317,159.802
C03238=1018.279,102.997,385.461,166.992,53.308,159.801
C03239=1018.284,103.246,385.443,166.995,53.301,159.800
C03240=1018.290,103.495,385.425,166.997,53.293,159.799
C03241=1018.295,103.745,385.407,167.000,53.285,159.798
C03242=1018.300,103.994,385.389,167.003,53.277,159.797
C03243=1018.305,104.243,385.371,167.006,53.269,159.796
C03244=1018.310,104.492,385.354,167.009,53.261,159.795
C03245=1018.316,104.742,385.335,167.011,53.253,159.794
C03246=1018.321,104.991,385.317,167.014,53.246,159.793
C03247=1018.326,105.240,385.299,167.018,53.237,159.792
C03248=1018.331,105.490,385.281,167.020,53.230,159.791
C03249=1018.336,105.739,385.264,167.023,53.222,159.790
C03250=1018.341,105.988,385.246,167.026,53.214,159.789
C03251=1018.347,106.237,385.228,167.028,53.206,159.788
C03252=1018.352,106.487,385.209,167.032,53.198,159.787
C03253=1018.357,106.769,385.190,167.035,53.189,159.786
C03254=1018.363,107.051,385.169,167.038,53.180,159.785
C03255=1018.369,107.334,385.148,167.041,53.171,159.784
C03256=1018.376,107.616,385.129,167.044,53.162,159.783
C03257=1018.381,107.865,385.110,167.047,53.154,159.782
C03258=1018.386,108.114,385.092,167.050,53.146,159.781
C03259=1018.391,108.363,385.074,167.053,53.138,159.780
C03260=1018.396,108.613,385.055,167.056,53.130,159.779
C03261=1018.402,108.862,385.038,167.058,53.122,159.778
C03262=1018.407,109.111,385.020,167.062,53.114,159.777
C03263=1018.412,109.360,385.002,167.064,53.106,159.776
C03264=1018.417,109.610,384.984,167.067,53.098,159.775
C03265=1018.422,109.860,384.965,167.070,53.090,159.774
C03266=1018.427,110.109,384.947,167.073,53.082,159.773
C03267=1018.433,110.358,384.929,167.076,53.074,159.772
C03268=1018.438,110.607,384.911,167.078,53.066,159.771
C03269=1018.443,110.856,384.893,167.081,53.059,159.770
C03270=1018.448,111.106,384.874,167.085,53.050,159.769
C03271=1018.454,111.355,384.856,167.087,53.042,159.768
C03272=1018.459,111.604,384.838,167.090,53.035,159.767
C03273=1018.463,111.853,384.820,167.092,53.027,159.766
C03274=1018.468,112.103,384.801,167.096,53.019,159.765
C03275=1018.474,112.352,384.783,167.099,53.011,159.764
C03276=1018.479,112.602,384.764,167.102,53.004,159.763
C03277=1018.483,112.851,384.746,167.104,52.996,159.762
C03278=1018.488,113.100,384.727,167.107,52.988,159.761
C03279=1018.494,113.350,384.708,167.110,52.981,159.760
C03280=1018.499,113.598,384.690,167.114,52.972,159.759
C03281=1018.504,113.848,384.671,167.116,52.965,159.758
C03282=1018.509,114.097,384.653,167.119,52.957,159.757
C03283=1018.514,114.346,384.634,167.121,52.949,159.756
C03284=1018.519,114.596,384.616,167.124,52.942,159.756
C03285=1018.524,114.845,384.597,167.127,52.934,159.755
C03286=1018.529,115.094,384.579,167.131,52.926,159.754
C03287=1018.534,115.343,384.560,167.133,52.918,159.753
C03288=1018.539,115.593,384.541,167.136,52.910,159.752
C03289=1018.544,115.842,384.523,167.139,52.903,159.751
C03290=1018.549,116.091,384.504,167.142,52.895,159.750
C03291=1018.555,116.340,384.485,167.145,52.887,159.749
C03292=1018.560,116.590,384.467,167.148,52.879,159.748
C03293=1018.565,116.838,384.448,167.151,52.871,159.747
C03294=1018.569,117.088,384.430,167.153,52.863,159.746
C03295=1018.575,117.337,384.411,167.156,52.856,159.745
C03296=1018.580,117.587,384.393,167.160,52.848,159.744
C03297=1018.585,117.835,384.374,167.163,52.840,159.743
C03298=1018.590,118.086,384.355,167.165,52.833,159.742
C03299=1018.595,118.334,384.336,167.168,52.825,159.741
C03300=1018.600,118.584,384.317,167.171,52.817,159.740
C03301=1018.607,118.940,384.291,167.176,52.805,159.739
C03302=1018.615,119.298,384.264,167.179,52.795,159.737
C03303=1018.622,119.654,384.237,167.183,52.783,159.736
C03304=1018.629,120.011,384.210,167.188,52.772,159.735
C03305=1018.634,120.261,384.191,167.191,52.764,159.734
C03306=1018.639,120.510,384.173,167.194,52.756,159.733
C03307=1018.644,120.759,384.154,167.197,52.748,159.732
C03308=1018.650,121.008,384.135,167.200,52.741,159.731
C03309=1018.655,121.258,384.116,167.203,52.733,159.730
C03310=1018.660,121.506,384.098,167.206,52.725,159.729
C03311=1018.666,121.756,384.078,167.209,52.717,159.728
C03312=1018.670,122.005,384.060,167.212,52.709,159.727
C03313=1018.675,122.217,384.044,167.214,52.703,159.726
C03314=1018.680,122.429,384.028,167.217,52.696,159.725
C03315=1018.683,122.641,384.012,167.220,52.689,159.725
C03316=1018.688,122.852,383.996,167.222,52.683,159.724
C03317=1018.692,123.065,383.980,167.224,52.676,159.723
C03318=1018.697,123.277,383.964,167.227,52.669,159.722
C03319=1018.701,123.488,383.948,167.230,52.663,159.721
C03320=1018.706,123.700,383.932,167.232,52.656,159.720
C03321=1018.711,123.949,383.913,167.236,52.648,159.719
C03322=1018.716,124.198,383.895,167.238,52.640,159.718
C03323=1018.721,124.448,383.875,167.241,52.632,159.717
C03324=1018.726,124.697,383.856,167.245,52.624,159.716
C03325=1018.731,124.947,383.838,167.247,52.616,159.715
C03326=1018.737,125.196,383.819,167.250,52.609,159.714
C03327=1018.742,125.444,383.800,167.254,52.600,159.714
C03328=1018.747,125.694,383.781,167.256,52.593,159.713
C03329=1018.752,125.943,383.763,167.259,52.585,159.712
C03330=1018.758,126.193,383.743,167.263,52.577,159.711
C03331=1018.763,126.441,383.724,167.265,52.569,159.710
C03332=1018.769,126.691,383.705,167.268,52.561,159.709
C03333=1018.773,126.940,383.687,167.272,52.553,159.708
C03334=1018.779,127.190,383.668,167.275,52.545,159.707
C03335=1018.784,127.438,383.649,167.278,52.538,159.706
C03336=1018.790,127.688,383.630,167.281,52.530,159.705
C03337=1018.795,127.936,383.611,167.284,52.522,159.704
C03338=1018.800,128.187,383.592,167.287,52.514,159.703
C03339=1018.805,128.436,383.573,167.290,52.506,159.702
C03340=1018.810,128.685,383.554,167.293,52.499,159.701
C03341=1018.815,128.934,383.535,167.296,52.491,159.700
C03342=1018.821,129.183,383.515,167.300,52.483,159.699
C03343=1018.826,129.433,383.497,167.302,52.475,159.698
C03344=1018.832,129.682,383.478,167.306,52.466,159.697
C03345=1018.837,129.931,383.459,167.309,52.459,159.696
C03346=1018.842,130.180,383.439,167.311,52.451,159.695
C03347=1018.847,130.429,383.420,167.314,52.443,159.694
C03348=1018.852,130.679,383.401,167.318,52.435,159.693
C03349=1018.857,130.928,383.382,167.321,52.428,159.692
C03350=1018.862,131.177,383.362,167.323,52.420,159.691
C03351=1018.867,131.426,383.343,167.327,52.412,159.691
C03352=1018.872,131.676,383.324,167.330,52.405,159.690
C03353=1018.877,131.925,383.304,167.333,52.397,159.689
C03354=1018.882,132.174,383.285,167.337,52.389,159.688
C03355=1018.887,132.423,383.266,167.339,52.381,159.687
C03356=1018.892,132.672,383.246,167.342,52.373,159.686
C03357=1018.897,132.922,383.227,167.345,52.366,159.685
C03358=1018.903,133.170,383.207,167.349,52.358,159.684
C03359=1018.909,133.420,383.188,167.352,52.350,159.683
C03360=1018.913,133.669,383.168,167.354,52.343,159.682
C03361=1018.919,133.918,383.149,167.358,52.335,159.681
C03362=1018.923,134.167,383.129,167.361,52.327,159.680
C03363=1018.929,134.417,383.110,167.364,52.319,159.679
C03364=1018.933,134.666,383.091,167.368,52.312,159.678
C03365=1018.939,134.915,383.072,167.371,52.304,159.677
C03366=1018.944,135.165,383.052,167.373,52.296,159.676
C03367=1018.949,135.413,383.032,167.377,52.288,159.675
C03368=1018.955,135.662,383.013,167.380,52.280,159.674
C03369=1018.959,135.912,382.993,167.383,52.273,159.673
C03370=1018.965,136.161,382.974,167.386,52.265,159.672
C03371=1018.970,136.411,382.954,167.389,52.257,159.672
C03372=1018.975,136.659,382.935,167.392,52.250,159.671
C03373=1018.980,136.909,382.915,167.396,52.242,159.670
C03374=1018.985,137.157,382.896,167.399,52.234,159.669
C03375=1018.990,137.407,382.876,167.401,52.226,159.668
C03376=1018.996,137.656,382.856,167.405,52.218,159.667
C03377=1019.000,137.905,382.837,167.408,52.210,159.666
C03378=1019.005,138.155,382.817,167.412,52.203,159.665
C03379=1019.011,138.404,382.798,167.415,52.195,159.664
C03380=1019.016,138.652,382.777,167.418,52.188,159.663
C03381=1019.022,138.935,382.755,167.421,52.179,159.662
C03382=1019.027,139.217,382.733,167.424,52.170,159.661
C03383=1019.033,139.499,382.711,167.429,52.162,159.660
C03384=1019.039,139.781,382.688,167.433,52.153,159.659
C03385=1019.044,140.031,382.668,167.435,52.145,159.658
C03386=1019.049,140.279,382.648,167.438,52.137,159.657
C03387=1019.054,140.529,382.628,167.442,52.130,159.656
C03388=1019.060,140.778,382.608,167.445,52.122,159.655
C03389=1019.064,141.027,382.589,167.448,52.115,159.654
C03390=1019.069,141.276,382.569,167.452,52.107,159.653
C03391=1019.075,141.525,382.549,167.454,52.099,159.652
C03392=1019.079,141.774,382.530,167.459,52.091,159.652
C03393=1019.085,142.023,382.509,167.461,52.084,159.651
C03394=1019.090,142.273,382.490,167.464,52.076,159.650
C03395=1019.095,142.521,382.470,167.468,52.068,159.649
C03396=1019.100,142.771,382.450,167.471,52.060,159.648
C03397=1019.105,143.020,382.429,167.474,52.053,159.647
C03398=1019.110,143.269,382.410,167.478,52.045,159.646
C03399=1019.116,143.518,382.390,167.481,52.038,159.645
C03400=1019.120,143.768,382.370,167.484,52.029,159.644
C03401=1019.126,144.017,382.350,167.487,52.022,159.643
C03402=1019.131,144.266,382.331,167.490,52.014,159.642
C03403=1019.136,144.515,382.310,167.494,52.007,159.642
C03404=1019.142,144.764,382.291,167.497,51.999,159.641
C03405=1019.147,145.013,382.270,167.501,51.991,159.640
C03406=1019.151,145.262,382.251,167.504,51.983,159.639
C03407=1019.157,145.511,382.230,167.506,51.976,159.638
C03408=1019.162,145.761,382.211,167.510,51.968,159.637
C03409=1019.168,146.010,382.190,167.513,51.961,159.636
C03410=1019.172,146.258,382.170,167.517,51.953,159.635
C03411=1019.177,146.508,382.150,167.520,51.945,159.634
C03412=1019.182,146.757,382.130,167.523,51.937,159.633
C03413=1019.188,147.006,382.109,167.527,51.930,159.632
C03414=1019.193,147.256,382.089,167.530,51.922,159.631
C03415=1019.197,147.505,382.069,167.533,51.914,159.630
C03416=1019.203,147.754,382.049,167.536,51.906,159.629
C03417=1019.208,148.003,382.029,167.540,51.899,159.629
C03418=1019.213,148.252,382.009,167.544,51.891,159.628
C03419=1019.218,148.501,381.989,167.546,51.884,159.627
C03420=1019.223,148.750,381.968,167.550,51.877,159.626
C03421=1019.228,149.000,381.948,167.553,51.869,159.625
C03422=1019.234,149.249,381.928,167.556,51.861,159.624
C03423=1019.239,149.498,381.907,167.560,51.853,159.623
C03424=1019.244,149.747,381.887,167.563,51.846,159.622
C03425=1019.248,149.996,381.867,167.566,51.838,159.621
C03426=1019.254,150.245,381.847,167.570,51.830,159.620
C03427=1019.259,150.494,381.826,167.573,51.823,159.619
C03428=1019.264,150.743,381.806,167.577,51.815,159.619
C03429=1019.269,150.992,381.785,167.580,51.808,159.618
C03430=1019.275,151.242,381.764,167.583,51.800,159.617
C03431=1019.279,151.491,381.745,167.586,51.792,159.616
C03432=1019.284,151.740,381.724,167.590,51.785,159.615
C03433=1019.290,151.989,381.704,167.594,51.777,159.614
C03434=1019.295,152.238,381.683,167.596,51.770,159.613
C03435=1019.300,152.487,381.663,167.600,51.762,159.612
C03436=1019.305,152.736,381.642,167.604,51.755,159.611
C03437=1019.311,152.985,381.622,167.607,51.747,159.611
C03438=1019.316,153.235,381.601,167.610,51.739,159.610
C03439=1019.321,153.483,381.581,167.613,51.732,159.609
C03440=1019.326,153.732,381.560,167.617,51.724,159.608
C03441=1019.330,153.982,381.540,167.620,51.716,159.607
C03442=1019.335,154.231,381.519,167.624,51.709,159.606
C03443=1019.340,154.480,381.499,167.627,51.701,159.605
C03444=1019.346,154.729,381.478,167.630,51.694,159.604
C03445=1019.352,155.011,381.454,167.635,51.685,159.603
C03446=1019.358,155.292,381.431,167.638,51.677,159.602
C03447=1019.363,155.575,381.408,167.642,51.668,159.601
C03448=1019.369,155.857,381.384,167.646,51.659,159.600
C03449=1019.374,156.106,381.363,167.650,51.652,159.599
C03450=1019.379,156.355,381.343,167.654,51.644,159.599
C03451=1019.385,156.604,381.322,167.656,51.636,159.597
C03452=1019.390,156.854,381.302,167.661,51.629,159.597
C03453=1019.395,157.103,381.281,167.664,51.622,159.596
C03454=1019.400,157.351,381.261,167.666,51.614,159.595
C03455=1019.404,157.601,381.240,167.671,51.607,159.594
C03456=1019.410,157.850,381.219,167.674,51.599,159.593
C03457=1019.415,158.099,381.199,167.677,51.591,159.592
C03458=1019.420,158.347,381.177,167.680,51.583,159.591
C03459=1019.426,158.596,381.157,167.685,51.576,159.591
C03460=1019.431,158.846,381.136,167.687,51.568,159.590
C03461=1019.435,159.095,381.115,167.692,51.561,159.589
C03462=1019.440,159.344,381.093,167.695,51.554,159.588
C03463=1019.446,159.593,381.073,167.698,51.547,159.587
C03464=1019.450,159.842,381.052,167.702,51.539,159.586
C03465=1019.456,160.091,381.030,167.705,51.532,159.585
C03466=1019.460,160.340,381.009,167.709,51.524,159.584
C03467=1019.465,160.589,380.987,167.712,51.517,159.584
C03468=1019.470,160.838,380.967,167.715,51.509,159.583
C03469=1019.475,161.088,380.946,167.719,51.502,159.582
C03470=1019.480,161.337,380.924,167.722,51.494,159.581
C03471=1019.485,161.586,380.903,167.727,51.487,159.580
C03472=1019.490,161.834,380.881,167.729,51.480,159.579
C03473=1019.495,162.084,380.861,167.733,51.473,159.578
C03474=1019.499,162.333,380.840,167.737,51.465,159.578
C03475=1019.504,162.582,380.818,167.740,51.458,159.577
C03476=1019.509,162.831,380.797,167.744,51.450,159.576
C03477=1019.514,163.080,380.775,167.747,51.443,159.575
C03478=1019.520,163.329,380.755,167.751,51.435,159.574
C03479=1019.524,163.578,380.733,167.754,51.428,159.573
C03480=1019.529,163.827,380.712,167.757,51.420,159.572
C03481=1019.534,164.076,380.691,167.762,51.413,159.572
C03482=1019.539,164.325,380.669,167.764,51.406,159.571
C03483=1019.545,164.574,380.648,167.769,51.398,159.570
C03484=1019.550,164.824,380.627,167.772,51.391,159.569
C03485=1019.554,165.073,380.605,167.776,51.384,159.568
C03486=1019.560,165.321,380.584,167.779,51.376,159.567
C03487=1019.565,165.570,380.562,167.783,51.369,159.567
C03488=1019.569,165.819,380.540,167.786,51.361,159.566
C03489=1019.575,166.068,380.520,167.790,51.354,159.565
C03490=1019.579,166.317,380.498,167.793,51.346,159.564
C03491=1019.585,166.566,380.478,167.798,51.339,159.563
C03492=1019.590,166.815,380.456,167.801,51.331,159.562
C03493=1019.594,167.064,380.434,167.805,51.324,159.562
C03494=1019.600,167.314,380.413,167.808,51.317,159.561
C03495=1019.605,167.563,380.391,167.812,51.309,159.560
C03496=1019.610,167.812,380.370,167.815,51.302,159.559
C03497=1019.615,168.061,380.349,167.819,51.295,159.558
C03498=1019.620,168.309,380.327,167.822,51.287,159.557
C03499=1019.625,168.558,380.306,167.827,51.280,159.557
C03500=1019.630,168.807,380.284,167.830,51.272,159.556
C03501=1019.635,169.057,380.262,167.834,51.265,159.555
C03502=1019.641,169.306,380.242,167.838,51.257,159.554
C03503=1019.646,169.555,380.220,167.841,51.250,159.553
C03504=1019.650,169.804,380.198,167.845,51.242,159.552
C03505=1019.656,170.053,380.177,167.849,51.235,159.551
C03506=1019.661,170.302,380.155,167.852,51.228,159.551
C03507=1019.667,170.551,380.134,167.856,51.221,159.550
C03508=1019.671,170.800,380.112,167.860,51.213,159.549
C03509=1019.677,171.082,380.088,167.864,51.205,159.548
C03510=1019.683,171.363,380.063,167.868,51.196,159.547
C03511=1019.688,171.645,380.039,167.872,51.187,159.546
C03512=1019.695,171.927,380.014,167.877,51.179,159.545
C03513=1019.700,172.176,379.993,167.880,51.172,159.544
C03514=1019.705,172.425,379.971,167.884,51.164,159.543
C03515=1019.709,172.673,379.950,167.888,51.156,159.543
C03516=1019.716,172.923,379.928,167.891,51.150,159.542
C03517=1019.720,173.171,379.906,167.895,51.142,159.541
C03518=1019.726,173.421,379.886,167.899,51.135,159.540
C03519=1019.731,173.669,379.864,167.903,51.127,159.539
C03520=1019.736,173.919,379.841,167.907,51.120,159.538
C03521=1019.742,174.167,379.820,167.910,51.112,159.537
C03522=1019.746,174.416,379.798,167.914,51.105,159.537
C03523=1019.752,174.666,379.776,167.918,51.097,159.536
C03524=1019.757,174.915,379.756,167.922,51.090,159.535
C03525=1019.762,175.164,379.734,167.926,51.082,159.534
C03526=1019.767,175.413,379.711,167.930,51.075,159.533
C03527=1019.773,175.662,379.690,167.933,51.068,159.532
C03528=1019.778,175.910,379.668,167.937,51.060,159.532
C03529=1019.783,176.160,379.646,167.941,51.053,159.531
C03530=1019.789,176.408,379.625,167.944,51.045,159.530
C03531=1019.793,176.657,379.603,167.949,51.038,159.529
C03532=1019.799,176.907,379.581,167.953,51.030,159.528
C03533=1019.804,177.155,379.559,167.956,51.023,159.527
C03534=1019.809,177.404,379.538,167.960,51.015,159.527
C03535=1019.815,177.654,379.515,167.964,51.008,159.526
C03536=1019.820,177.902,379.494,167.968,51.000,159.525
C03537=1019.826,178.152,379.472,167.971,50.993,159.524
C03538=1019.831,178.400,379.451,167.976,50.986,159.523
C03539=1019.836,178.649,379.429,167.980,50.978,159.522
C03540=1019.842,178.898,379.407,167.983,50.971,159.522
C03541=1019.847,179.147,379.385,167.987,50.963,159.521
C03542=1019.852,179.397,379.363,167.991,50.956,159.520
C03543=1019.857,179.645,379.341,167.995,50.948,159.519
C03544=1019.863,179.894,379.320,167.999,50.941,159.518
C03545=1019.868,180.143,379.298,168.003,50.933,159.517
C03546=1019.873,180.392,379.276,168.007,50.926,159.517
C03547=1019.879,180.641,379.254,168.011,50.918,159.516
C03548=1019.884,180.890,379.232,168.015,50.910,159.515
C03549=1019.890,181.140,379.210,168.018,50.904,159.514
C03550=1019.895,181.388,379.189,168.022,50.896,159.513
C03551=1019.901,181.638,379.167,168.027,50.889,159.513
C03552=1019.906,181.886,379.144,168.031,50.881,159.512
C03553=1019.911,182.135,379.122,168.034,50.874,159.511
C03554=1019.916,182.384,379.100,168.039,50.867,159.510
C03555=1019.921,182.634,379.078,168.043,50.859,159.509
C03556=1019.926,182.882,379.054,168.046,50.852,159.508
C03557=1019.931,183.132,379.032,168.050,50.845,159.508
C03558=1019.936,183.380,379.010,168.055,50.838,159.507
C03559=1019.941,183.630,378.987,168.058,50.830,159.506
C03560=1019.946,183.878,378.964,168.062,50.823,159.505
C03561=1019.951,184.127,378.942,168.066,50.816,159.505
C03562=1019.957,184.376,378.919,168.070,50.809,159.504
C03563=1019.961,184.625,378.897,168.074,50.802,159.503
C03564=1019.966,184.874,378.874,168.077,50.795,159.502
C03565=1019.971,185.123,378.852,168.082,50.788,159.501
C03566=1019.976,185.372,378.829,168.086,50.780,159.501
C03567=1019.981,185.621,378.807,168.090,50.774,159.500
C03568=1019.987,185.869,378.784,168.094,50.766,159.499
C03569=1019.991,186.119,378.761,168.098,50.759,159.498
C03570=1019.997,186.368,378.738,168.101,50.752,159.498
C03571=1020.001,186.616,378.717,168.106,50.745,159.497
C03572=1020.006,186.866,378.693,168.110,50.738,159.496
C03573=1020.013,187.146,378.668,168.114,50.729,159.495
C03574=1020.018,187.428,378.642,168.119,50.721,159.494
C03575=1020.024,187.709,378.616,168.124,50.713,159.494
C03576=1020.030,187.990,378.590,168.128,50.705,159.493
C03577=1020.035,188.240,378.568,168.133,50.698,159.492
C03578=1020.040,188.488,378.545,168.137,50.691,159.491
C03579=1020.045,188.738,378.523,168.140,50.683,159.490
C03580=1020.050,188.986,378.500,168.144,50.676,159.490
C03581=1020.056,189.235,378.477,168.149,50.669,159.489
C03582=1020.061,189.484,378.454,168.153,50.662,159.488
C03583=1020.066,189.733,378.432,168.157,50.654,159.487
C03584=1020.071,189.982,378.409,168.161,50.647,159.486
C03585=1020.076,190.230,378.386,168.165,50.640,159.486
C03586=1020.081,190.480,378.363,168.170,50.633,159.485
C03587=1020.087,190.729,378.340,168.174,50.626,159.484
C03588=1020.092,190.977,378.318,168.177,50.619,159.483
C03589=1020.097,191.226,378.294,168.181,50.611,159.483
C03590=1020.102,191.475,378.272,168.186,50.604,159.482
C03591=1020.108,191.724,378.250,168.190,50.597,159.481
C03592=1020.113,191.973,378.226,168.195,50.590,159.481
C03593=1020.118,192.222,378.203,168.198,50.583,159.479
C03594=1020.123,192.470,378.180,168.202,50.576,159.479
C03595=1020.128,192.720,378.158,168.207,50.569,159.478
C03596=1020.134,192.969,378.135,168.211,50.561,159.477
C03597=1020.139,193.217,378.112,168.215,50.554,159.476
C03598=1020.144,193.466,378.089,168.220,50.547,159.476
C03599=1020.150,193.715,378.066,168.223,50.540,159.475
C03600=1020.155,193.964,378.043,168.228,50.533,159.474
C03601=1020.160,194.213,378.020,168.232,50.526,159.474
C03602=1020.165,194.462,377.997,168.236,50.518,159.473
C03603=1020.171,194.711,377.974,168.240,50.511,159.472
C03604=1020.175,194.959,377.951,168.245,50.504,159.471
C03605=1020.181,195.208,377.928,168.249,50.497,159.471
C03606=1020.187,195.457,377.905,168.254,50.490,159.470
C03607=1020.192,195.706,377.882,168.257,50.483,159.469
C03608=1020.198,195.955,377.859,168.261,50.475,159.468
C03609=1020.203,196.203,377.836,168.266,50.468,159.467
C03610=1020.208,196.453,377.813,168.270,50.461,159.467
C03611=1020.213,196.702,377.790,168.275,50.454,159.466
C03612=1020.219,196.950,377.767,168.279,50.447,159.465
C03613=1020.224,197.200,377.743,168.283,50.439,159.464
C03614=1020.229,197.448,377.721,168.288,50.432,159.464
C03615=1020.235,197.697,377.698,168.292,50.425,159.463
C03616=1020.240,197.946,377.674,168.297,50.418,159.462
C03617=1020.246,198.195,377.651,168.301,50.411,159.462
C03618=1020.251,198.444,377.628,168.305,50.403,159.461
C03619=1020.256,198.693,377.605,168.309,50.396,159.460
C03620=1020.262,198.941,377.582,168.313,50.389,159.459
C03621=1020.267,199.190,377.559,168.318,50.382,159.459
C03622=1020.272,199.439,377.536,168.322,50.375,159.458
C03623=1020.277,199.688,377.512,168.326,50.368,159.457
C03624=1020.283,199.937,377.488,168.331,50.361,159.456
C03625=1020.288,200.186,377.465,168.335,50.354,159.456
C03626=1020.293,200.435,377.441,168.340,50.347,159.455
C03627=1020.299,200.684,377.418,168.344,50.340,159.454
C03628=1020.304,200.932,377.395,168.349,50.333,159.454
C03629=1020.309,201.181,377.371,168.353,50.326,159.453
C03630=1020.314,201.430,377.347,168.357,50.319,159.452
C03631=1020.320,201.679,377.324,168.361,50.312,159.451
C03632=1020.325,201.928,377.300,168.366,50.305,159.451
C03633=1020.330,202.176,377.276,168.370,50.298,159.450
C03634=1020.336,202.425,377.253,168.375,50.291,159.449
C03635=1020.341,202.674,377.230,168.379,50.284,159.449
C03636=1020.346,202.923,377.205,168.384,50.277,159.448
C03637=1020.368,203.963,377.107,168.833,50.371,159.543
